				3: (* Wait Z move done *)
				   IF GV_Axes.stAxisZ.bAutoDone THEN
						GV_Axes.stAxisZ.bAutoCmdAbs:=FALSE;
						(*Log*)
							PRG_Log_WM.fbLogWM.M_Write_Log('FB_11_Action_ToolMagazineCheckAll : 2_MoveLocation : 3 : Z move done');
						iSubStep:=4; // Next SubStep
					ELSIF GV_Axes.stAxisZ.stDriveAx8206.AxisRef.Status.Error OR GV_Axes.stAxisZ.stDriveAx8206.AxisRef.Status.ErrorStop OR GV_Axes.stAxisZ.stDriveAx8206.AxisRef.Status.ErrorID<>0 THEN
						bError:=TRUE;
						udiErrorID:=231; // 231 = Step 2 SubStep 3 Error Axis Z 1
						GV_Axes.stAxisZ.bAutoCmdAbs:=FALSE;
						tonTimeout.IN:=FALSE;
						(*Log*)
							PRG_Log_WM.fbLogWM.M_Write_Log('FB_11_Action_ToolMagazineCheckAll : 2_MoveLocation=Error');
							PRG_Log_WM.fbLogWM.M_Write_Log(CONCAT('FB_11_Action_ToolMagazineCheckAll : ErrorID=',UDINT_TO_STRING(udiErrorID)));
						iSubStep:=0; // Stop SubStep
						iStep:=0; // Idle Step
					END_IF

				4: (* Start Y move *)
					GV_Axes.stAxisY.lrAutoPosAbs:=GV_Tool_Magazine.aCheckLocation[iLocation].lrYcoord;
					GV_Axes.stAxisY.bAutoCmdAbs:=TRUE;
					(*Log*)
						PRG_Log_WM.fbLogWM.M_Write_Log('FB_11_Action_ToolMagazineCheckAll : 2_MoveLocation : 4 : Start Y move');
					iSubStep:=5; // Next Step

				5: (* Wait Y move done *)
				   IF GV_Axes.stAxisY.bAutoDone THEN
						GV_Axes.stAxisY.bAutoCmdAbs:=FALSE;
						(*Log*)
							PRG_Log_WM.fbLogWM.M_Write_Log('FB_11_Action_ToolMagazineCheckAll : 2_MoveLocation : 5 : Y move done');
							PRG_Log_WM.fbLogWM.M_Write_Log('FB_11_Action_ToolMagazineCheckAll : 2_MoveLocation->3_Check');
						iSubStep:=0; // End SubStep
						iStep:=3; // Next Step
					ELSIF GV_Axes.stAxisY.stDriveAx8206.AxisRef.Status.Error OR GV_Axes.stAxisY.stDriveAx8206.AxisRef.Status.ErrorStop OR GV_Axes.stAxisY.stDriveAx8206.AxisRef.Status.ErrorID<>0 THEN
						bError:=TRUE;
						udiErrorID:=251; // 251 = Step 2 SubStep 5 Error Axis Y 1
						GV_Axes.stAxisY.bAutoCmdAbs:=FALSE;
						tonTimeout.IN:=FALSE;
						(*Log*)
							PRG_Log_WM.fbLogWM.M_Write_Log('FB_11_Action_ToolMagazineCheckAll : 2_MoveLocation=Error');
							PRG_Log_WM.fbLogWM.M_Write_Log(CONCAT('FB_11_Action_ToolMagazineCheckAll : ErrorID=',UDINT_TO_STRING(udiErrorID)));
						iSubStep:=0; // Stop SubStep
						iStep:=0; // Idle Step
					END_IF

				8: (* Start Y home move *)
					GV_Axes.stAxisY.lrAutoPosAbs:=GV_Tool_Magazine.stManipulator.lrYHome;
					GV_Axes.stAxisY.bAutoCmdAbs:=TRUE;
					(*Log*)
						PRG_Log_WM.fbLogWM.M_Write_Log('FB_11_Action_ToolMagazineCheckAll : 2_MoveLocation : 8 : Start Y home move');
					iSubStep:=9; // Next SubStep

				9: (* Wait Y home move done *)
				   IF GV_Axes.stAxisY.bAutoDone THEN
						GV_Axes.stAxisY.bAutoCmdAbs:=FALSE;
						(*Log*)
							PRG_Log_WM.fbLogWM.M_Write_Log('FB_11_Action_ToolMagazineCheckAll : 2_MoveLocation : 9 : Y home move done');
						iSubStep:=0; // End SubStep
					ELSIF GV_Axes.stAxisY.stDriveAx8206.AxisRef.Status.Error OR GV_Axes.stAxisY.stDriveAx8206.AxisRef.Status.ErrorStop OR GV_Axes.stAxisY.stDriveAx8206.AxisRef.Status.ErrorID<>0 THEN
						bError:=TRUE;
						udiErrorID:=291; // 291 = Step 2 SubStep 9 Error Axis Y 1
						GV_Axes.stAxisY.bAutoCmdAbs:=FALSE;
						tonTimeout.IN:=FALSE;
						(*Log*)
							PRG_Log_WM.fbLogWM.M_Write_Log('FB_11_Action_ToolMagazineCheckAll : 2_MoveLocation=Error');
							PRG_Log_WM.fbLogWM.M_Write_Log(CONCAT('FB_11_Action_ToolMagazineCheckAll : ErrorID=',UDINT_TO_STRING(udiErrorID)));
						iSubStep:=0; // Stop SubStep
						iStep:=0; // Idle Step
					END_IF

				END_CASE
				
				IF tonTimeout.Q THEN
					bError:=TRUE;
					udiErrorID:=299; // 299 = Step 2 Error Timeout 99
					GV_Axes.stAxisX.bAutoCmdAbs:=FALSE;
					GV_Axes.stAxisZ.bAutoCmdAbs:=FALSE;
					GV_Axes.stAxisY.bAutoCmdAbs:=FALSE;
					tonTimeout.IN:=FALSE;
					(*Log*)
						PRG_Log_WM.fbLogWM.M_Write_Log('FB_11_Action_ToolMagazineCheckAll : 2_MoveLocation : Error');
						PRG_Log_WM.fbLogWM.M_Write_Log(CONCAT('FB_11_Action_ToolMagazineCheckAll : ErrorID = ',UDINT_TO_STRING(udiErrorID)));
					iSubStep:=0; // Stop SubStep
					iStep:=0; // Idle Step
				END_IF
	
			3: (* Step 3 = Check Tool presence in Location *)
				(*Conversion*)
					lrToolPresenceRack:=(INT_TO_LREAL(GV_IO.aiToolPresenceRack))*(2/32767); //(0..10V) = (0..32767) = (0..2mm)
				(*Tolerance*)
					IF lrToolPresenceRack>=(lrToolDistance-lrToolDistanceTolerance) AND lrToolPresenceRack<=(lrToolDistance+lrToolDistanceTolerance) THEN
						bToleranceOK:=TRUE;
					ELSE
						bToleranceOK:=FALSE;
					END_IF
				(*Check*)
					IF bToleranceOK THEN
						(*Update*)
							GV_Tool_Magazine.aCheckLocation[iLocation].bToolPresence:=TRUE; // OK
						(*Log*)
							strTextLog:=INT_TO_STRING(GV_IO.aiToolPresenceRack);
							PRG_Log_WM.fbLogWM.M_Write_Log(CONCAT('FB_11_Action_ToolMagazineCheckAll : 3_Check : Sensor in INT = ',strTextLog));
							strTextLog:=LREAL_TO_STRING(lrToolPresenceRack);
							PRG_Log_WM.fbLogWM.M_Write_Log(CONCAT('FB_11_Action_ToolMagazineCheckAll : 3_Check : Sensor in LREAL(mm) = ',strTextLog));
							PRG_Log_WM.fbLogWM.M_Write_Log('FB_11_Action_ToolMagazineCheckAll : 3_Check : Tolerance = OK');						
						bToleranceOK:=FALSE;	
						lrToolPresenceRack:=0.0;
						iStep:=4; // Next Step
					ELSE
						(*Update*)
							GV_Tool_Magazine.aCheckLocation[iLocation].bToolPresence:=FALSE; // NOK
						(*Log*)
							strTextLog:=INT_TO_STRING(GV_IO.aiToolPresenceRack);
							PRG_Log_WM.fbLogWM.M_Write_Log(CONCAT('FB_11_Action_ToolMagazineCheckAll : 3_Check : Sensor in INT = ',strTextLog));
							strTextLog:=LREAL_TO_STRING(lrToolPresenceRack);
							PRG_Log_WM.fbLogWM.M_Write_Log(CONCAT('FB_11_Action_ToolMagazineCheckAll : 3_Check : Sensor in LREAL(mm) = ',strTextLog));
							PRG_Log_WM.fbLogWM.M_Write_Log('FB_11_Action_ToolMagazineCheckAll : 3_Check : Tolerance = NOK');						
						bToleranceOK:=FALSE;	
						lrToolPresenceRack:=0.0;
						iStep:=4; // Next Step
					END_IF
			
			4: (* Step 4 = Next Location Or End *)
				iLocation:=iLocation+1;
				IF iLocation>(GV_Tool_Magazine.iCheckLocationTopSize+GV_Tool_Magazine.iCheckLocationBottomSize) THEN
					(*Log*)
						PRG_Log_WM.fbLogWM.M_Write_Log('FB_11_Action_ToolMagazineCheckAll: End : 4_NextEnd->5_Tunnel');
					iStep:=5; // Next Step = End
				ELSE
					(*Log*)
						PRG_Log_WM.fbLogWM.M_Write_Log('FB_11_Action_ToolMagazineCheckAll : Next : 4_NextEnd->1_Tunnel');
					iStep:=1; // Next Step = Next Location
				END_IF
		(* End Check sequence *)

		5: (* Step 5 = Tunnel passage (if needed) *)
			IF (NOT bTunnelTravel) THEN
				IF GV_Tool_Magazine.stManipulator.ePositionMag=ENUM_Position_Magazine.Top THEN
					bTunnelTravel:=FALSE;
					(*Log*)
						PRG_Log_WM.fbLogWM.M_Write_Log('FB_11_Action_ToolMagazineCheckAll : 5_Tunnel : No Need to Travel');
						PRG_Log_WM.fbLogWM.M_Write_Log('FB_11_Action_ToolMagazineCheckAll : 5_Tunnel->6_PositionHome');
					iSubStep:=0; // For next Step
					iStep:=6; // Next Step
				END_IF	
				IF GV_Tool_Magazine.stManipulator.ePositionMag=ENUM_Position_Magazine.Bottom THEN
					eTunnelMode:=ENUM_Tunnel_MODE.BottomToTop;
					bTunnelTravel:=TRUE;
					(*Log*)
						PRG_Log_WM.fbLogWM.M_Write_Log('FB_11_Action_ToolMagazineCheckAll : 5_Tunnel : Need to Travel Bottom->Top');
				END_IF			
				IF GV_Tool_Magazine.stManipulator.ePositionMag=ENUM_Position_Magazine.Unknow THEN // Manipulator Unknow position
					bError:=TRUE;
					udiErrorID:=501; // 501 = Step 5 Error Tunnel 01
					fbTunnel.bStart:=FALSE;
					bTunnelTravel:=FALSE;
					(*Log*)
						PRG_Log_WM.fbLogWM.M_Write_Log('FB_11_Action_ToolMagazineCheckAll : 5_Tunnel=Error');
						PRG_Log_WM.fbLogWM.M_Write_Log(CONCAT('FB_11_Action_ToolMagazineCheckAll : ErrorID=',UDINT_TO_STRING(udiErrorID)));
					iStep:=0; // Idle Step
				END_IF
			END_IF
			
			IF bTunnelTravel AND (NOT fbTunnel.bStart) AND (NOT fbTunnel.bBusy) THEN // Tunnel Start
				fbTunnel.bStart:=TRUE;
			END_IF
			IF fbTunnel.bDone THEN // Tunnel Done
				fbTunnel.bStart:=FALSE;
				bTunnelTravel:=FALSE;
				(*Log*)
					PRG_Log_WM.fbLogWM.M_Write_Log('FB_11_Action_ToolMagazineCheckAll : 5_Tunnel->6_PositionHome');
				iSubStep:=0; // For next Step
				iStep:=6; // Next Step
			ELSIF fbTunnel.bError THEN // Tunnel Error
				bError:=TRUE;
				udiErrorID:=500+fbTunnel.udiErrorID; // 5xx = Step 5 Error + Error xx fbTunnel
				fbTunnel.bStart:=FALSE;
				bTunnelTravel:=FALSE;
				(*Log*)
					PRG_Log_WM.fbLogWM.M_Write_Log('FB_11_Action_ToolMagazineCheckAll : 5_Tunnel=Error');
					PRG_Log_WM.fbLogWM.M_Write_Log(CONCAT('FB_11_Action_ToolMagazineCheckAll : ErrorID=',UDINT_TO_STRING(udiErrorID)));
				iStep:=0; // Idle Step
			END_IF
			
			IF tonTimeout.Q THEN
				bError:=TRUE;
				udiErrorID:=599; // 599 = Step 5 Error Timeout 99
				fbTunnel.bStart:=FALSE;
				bTunnelTravel:=FALSE;
				tonTimeout.IN:=FALSE;
				(*Log*)
					PRG_Log_WM.fbLogWM.M_Write_Log('FB_11_Action_ToolMagazineCheckAll : 5_Tunnel : Error');
					PRG_Log_WM.fbLogWM.M_Write_Log(CONCAT('FB_11_Action_ToolMagazineCheckAll : ErrorID = ',UDINT_TO_STRING(udiErrorID)));
				iSubStep:=0; // Stop SubStep
				iStep:=0; // Idle Step
			END_IF
				
		6: (* Step 6 = Home Position*)
		
			CASE iSubStep OF //Y->X->Z

				0: (* Start Y home move *)
					GV_Axes.stAxisY.lrAutoPosAbs:=GV_Tool_Magazine.stManipulator.lrYHome;
					GV_Axes.stAxisY.bAutoCmdAbs:=TRUE;
					(*Log*)
						PRG_Log_WM.fbLogWM.M_Write_Log('FB_11_Action_ToolMagazineCheckAll : 6_PositionHome : 0 : Start Y home move');
					iSubStep:=1; // Next Step
				
				1: (* Wait Y home move done *)
					IF GV_Axes.stAxisY.bAutoDone THEN
						GV_Axes.stAxisY.bAutoCmdAbs:=FALSE;
						(*Log*)
							PRG_Log_WM.fbLogWM.M_Write_Log('FB_11_Action_ToolMagazineCheckAll : 6_PositionHome : 1 : Y move done');
						iSubStep:=2; // Next SubStep
					ELSIF GV_Axes.stAxisY.stDriveAx8206.AxisRef.Status.Error OR GV_Axes.stAxisY.stDriveAx8206.AxisRef.Status.ErrorStop OR GV_Axes.stAxisY.stDriveAx8206.AxisRef.Status.ErrorID<>0 THEN
						bError:=TRUE;
						udiErrorID:=611; // 611 = Step 6 SubStep 1 Error Axis Y 1
						GV_Axes.stAxisY.bAutoCmdAbs:=FALSE;
						tonTimeout.IN:=FALSE;
						(*Log*)
							PRG_Log_WM.fbLogWM.M_Write_Log('FB_11_Action_ToolMagazineCheckAll : 6_PositionHome=Error');
							PRG_Log_WM.fbLogWM.M_Write_Log(CONCAT('FB_11_Action_ToolMagazineCheckAll : ErrorID=',UDINT_TO_STRING(udiErrorID)));
						iSubStep:=0; // Stop SubStep
						iStep:=0; // Idle Step
					END_IF
				
				2: (* Start X home move *)
					GV_Axes.stAxisX.lrAutoPosAbs:=GV_Tool_Magazine.stManipulator.lrXHome;
					GV_Axes.stAxisX.bAutoCmdAbs:=TRUE;
					(*Log*)
						PRG_Log_WM.fbLogWM.M_Write_Log('FB_11_Action_ToolMagazineCheckAll : 6_PositionHome : 2 : Start X home move');
					iSubStep:=3; // Next Step
					
				3: (* Wait X home move done *)
					IF GV_Axes.stAxisX.bAutoDone THEN
						GV_Axes.stAxisX.bAutoCmdAbs:=FALSE;
						(*Log*)
							PRG_Log_WM.fbLogWM.M_Write_Log('FB_11_Action_ToolMagazineCheckAll : 6_PositionHome : 3 : X move done');
						iSubStep:=4; // Next SubStep
					ELSIF GV_Axes.stAxisX.stDriveAx8206.AxisRef.Status.Error OR GV_Axes.stAxisX.stDriveAx8206.AxisRef.Status.ErrorStop OR GV_Axes.stAxisX.stDriveAx8206.AxisRef.Status.ErrorID<>0 THEN
						bError:=TRUE;
						udiErrorID:=631; // 631 = Step 6 SubStep 3 Error Axis X 1
						GV_Axes.stAxisX.bAutoCmdAbs:=FALSE;
						tonTimeout.IN:=FALSE;
						(*Log*)
							PRG_Log_WM.fbLogWM.M_Write_Log('FB_11_Action_ToolMagazineCheckAll : 6_PositionHome=Error');
							PRG_Log_WM.fbLogWM.M_Write_Log(CONCAT('FB_11_Action_ToolMagazineCheckAll : ErrorID=',UDINT_TO_STRING(udiErrorID)));
						iSubStep:=0; // Stop SubStep
						iStep:=0; // Idle Step
					END_IF
				
				4: (* Start Z home move *)
					GV_Axes.stAxisZ.lrAutoPosAbs:=GV_Tool_Magazine.stManipulator.lrZHome;
					GV_Axes.stAxisZ.bAutoCmdAbs:=TRUE;
					(*Log*)
						PRG_Log_WM.fbLogWM.M_Write_Log('FB_11_Action_ToolMagazineCheckAll : 6_PositionHome : 4 : Start X home move');
					iSubStep:=5; // Next Step
					
				5: (* Wait Z home move done *)
					IF GV_Axes.stAxisZ.bAutoDone THEN
						GV_Axes.stAxisZ.bAutoCmdAbs:=FALSE;
						(*Log*)
							PRG_Log_WM.fbLogWM.M_Write_Log('FB_11_Action_ToolMagazineCheckAll : 6_PositionHome : 5 : Y move done');
							PRG_Log_WM.fbLogWM.M_Write_Log('FB_11_Action_ToolMagazineCheckAll : 6_PositionHome->0_Idle');
						tonTimeout.IN:=FALSE;
						iSubStep:=0; // End SubStep
						iStep:=0; // End Step
						bDone:=TRUE;
						bBusy:=FALSE;
					ELSIF GV_Axes.stAxisZ.stDriveAx8206.AxisRef.Status.Error OR GV_Axes.stAxisZ.stDriveAx8206.AxisRef.Status.ErrorStop OR GV_Axes.stAxisZ.stDriveAx8206.AxisRef.Status.ErrorID<>0 THEN
						bError:=TRUE;
						udiErrorID:=651; // 651 = Step 6 SubStep 5 Error Axis Z 1
						GV_Axes.stAxisZ.bAutoCmdAbs:=FALSE;
						tonTimeout.IN:=FALSE;
						(*Log*)
							PRG_Log_WM.fbLogWM.M_Write_Log('FB_11_Action_ToolMagazineCheckAll : 6_PositionHome=Error');
							PRG_Log_WM.fbLogWM.M_Write_Log(CONCAT('FB_11_Action_ToolMagazineCheckAll : ErrorID=',UDINT_TO_STRING(udiErrorID)));
						iSubStep:=0; // Stop SubStep
						iStep:=0; // Idle Step
					END_IF
					
			END_CASE
				
			IF tonTimeout.Q AND tonTimeout.PT<>T#0S THEN
				bError:=TRUE;
				udiErrorID:=699; // 699 = Step 6 Error Timeout 99
				GV_Axes.stAxisX.bAutoCmdAbs:=FALSE;
				GV_Axes.stAxisZ.bAutoCmdAbs:=FALSE;
				GV_Axes.stAxisY.bAutoCmdAbs:=FALSE;
				tonTimeout.IN:=FALSE;
				(*Log*)
					PRG_Log_WM.fbLogWM.M_Write_Log('FB_11_Action_ToolMagazineCheckAll : 6_PositionHome : Error');
					PRG_Log_WM.fbLogWM.M_Write_Log(CONCAT('FB_11_Action_ToolMagazineCheckAll : ErrorID = ',UDINT_TO_STRING(udiErrorID)));
				iSubStep:=0; // Stop SubStep
				iStep:=0; // Idle Step
			END_IF

	END_CASE

END_FUNCTION_BLOCK

// ---- 08_Cycle/03_POUs/02_FBs/FB_200_Action_HomePosition.TcPOU
FUNCTION_BLOCK FB_200_Action_HomePosition
VAR_INPUT
	(** SETUP ST **)
		
	(** SETUP TIME **)
		(*Tunnel*)
			tTunnelTimeout : TIME ; // Value of the timeout for travel the tunnel
		(* Step x *)
			tMovexTimeout : TIME ; // Value of the timeout for Step x

	(** SETUP LREAL **)

	(** SETUP FLAG **)
			
	(** PROCESS FLAG **)
	    bInit : BOOL ; // Init the Fb
	    bStart : BOOL ; // Start the Fb
END_VAR
VAR_OUTPUT
	(** PROCESS UDINT **)
		udiErrorID : UDINT ; // Fb Error ID
		
	(** PROCESS FLAG **)
		bBusy  : BOOL ; // Fb is Busy
		bDone  : BOOL ; // Fb is Done
		bError : BOOL ; // Fb in Error
END_VAR
VAR_IN_OUT
END_VAR	
VAR
	(** SETUP ENUM **)
		(*Tunnel*)
			eTunnelMode : ENUM_Tunnel_Mode; // Tunnel mode for travel (fbTunnel)

	(** SETUP TIME **)
	
	(** SETUP FLAG **)
		
	(** PROCESS STRING **)
		strTextLog : STRING ; // Text to Log
		
	(** PROCESS LREAL **)
		
	(** PROCESS INT **)
		iStep  : INT := 0 ; // Step of the Fb
		iSubStep : INT := 0 ; // SubStep of the Fb
		iPrevStep : INT := 0 ; // Previous Step of the Fb
		iPrevSubStep : INT := 0 ; // Previous Subtep of the Fb
		
	(** PROCESS FLAG + R_TRIG **)
		rtInit : R_TRIG ; // FB Init at rising edge
		rtStart : R_TRIG ; // FB Start at rising edge
		(*Tunnel*)
			bTunnelTravel : BOOL ; // Need to travel the tunnel
				
	(** FB **)
		(*Tunnel*)
			fbTunnel : FB_Manipulator_Tunnel ;
		(* Step x *)
			tonTimeoutMovex : TON ; // TON timeout for the Step x
END_VAR

//-----------------------------------------------------------------------------------------
//
//                  			FB_200_Action_HomePosition
//
//		ESSAI		Management of move to home position (Manipulator only)
//-----------------------------------------------------------------------------------------
//
//Auteur: G.GOETZ
//Création: 01.04.2026
//Dernière modification : 01.04.2026 (G.GOETZ)
//       			
//-----------------------------------------------------------------------------------------
//
//     							Liste des modifications  	
//
// 01.04.2026 (G.GOETZ) -> Création		
//-----------------------------------------------------------------------------------------

(** FB CALL **)
	rtInit(CLK:=bInit);
	rtStart(CLK:=bStart);
		
	tonTimeoutMovex();
	fbTunnel( // Call Tunnel travel
			eTunnelMode:=eTunnelMode,
			tTimeout:=tTunnelTimeout
			);

(** INIT **)
	IF (rtinit.Q OR bInit) AND (NOT bStart) THEN
		bBusy:=FALSE;
		bDone:=FALSE;
		bError:=FALSE;
		udiErrorID:=0;
		iStep:=0;
		iSubStep:=0;
		bInit:=FALSE;
	END_IF

(** STEPS **)
    CASE iStep OF
		
        0: (* Step 0 = Idle + Check *)
            bBusy:=FALSE;
            bDone:=FALSE;
			bError:=FALSE;
			udiErrorID:=0;
			iSubStep:=0;
			
			tonTimeoutMovex.IN:=FALSE;
			
			bTunnelTravel:=FALSE;
			
			(* Idle->Start *)
				IF rtStart.Q AND (NOT bInit) THEN
					bBusy:=TRUE;
					(*Log*)
						PRG_Log_WM.fbLogWM.M_Write_Log('FB_200_Action_HomePosition : 0_Idle : Manipulator to Home Position');
						PRG_Log_WM.fbLogWM.M_Write_Log('FB_200_Action_HomePosition : 0_Idle->1_Tunnel');
					iStep:=1;
				END_IF
				
		1: (* Step 1 = Tunnel passage (if needed) *)
			IF (NOT bTunnelTravel) THEN
				IF GV_Tool_Magazine.stManipulator.ePositionMag=ENUM_Position_Magazine.Top THEN
					bTunnelTravel:=FALSE;
					(*Log*)
						PRG_Log_WM.fbLogWM.M_Write_Log('FB_200_Action_HomePosition : 1_Tunnel : No Need to Travel');
						PRG_Log_WM.fbLogWM.M_Write_Log('FB_200_Action_HomePosition : 1_Tunnel->2_MoveHome');
					iStep:=2; // Next Step
				END_IF	
				IF GV_Tool_Magazine.stManipulator.ePositionMag=ENUM_Position_Magazine.Bottom THEN
					eTunnelMode:=ENUM_Tunnel_MODE.BottomToTop;
					bTunnelTravel:=TRUE;
					(*Log*)
						PRG_Log_WM.fbLogWM.M_Write_Log('FB_200_Action_HomePosition : 1_Tunnel : Need to Travel Bottom->Top');
				END_IF			
				IF GV_Tool_Magazine.stManipulator.ePositionMag=ENUM_Position_Magazine.Unknow THEN // Manipulator Unknow position
					bError:=TRUE;
					udiErrorID:=101; // 101 = Step 1 Error Tunnel 01
					fbTunnel.bStart:=FALSE;
					bTunnelTravel:=FALSE;
					(*Log*)
						PRG_Log_WM.fbLogWM.M_Write_Log('FB_200_Action_HomePosition : 1_Tunnel=Error');
						PRG_Log_WM.fbLogWM.M_Write_Log(CONCAT('FB_200_Action_HomePosition : ErrorID=',UDINT_TO_STRING(udiErrorID)));
					iStep:=0; // Idle Step
				END_IF
			END_IF
			
			IF bTunnelTravel AND (NOT fbTunnel.bStart) AND (NOT fbTunnel.bBusy) THEN // Tunnel Start
				fbTunnel.bStart:=TRUE;
			END_IF
			IF fbTunnel.bDone THEN // Tunnel Done
				fbTunnel.bStart:=FALSE;
				bTunnelTravel:=FALSE;
				(*Log*)
					PRG_Log_WM.fbLogWM.M_Write_Log('FB_200_Action_HomePosition : 1_Tunnel->2_MoveHome');
				iStep:=2; // Next Step
			ELSIF fbTunnel.bError THEN // Tunnel Error
				bError:=TRUE;
				udiErrorID:=100+fbTunnel.udiErrorID; // 1xx = Step 1 Error + Error xx fbTunnel
				fbTunnel.bStart:=FALSE;
				bTunnelTravel:=FALSE;
				(*Log*)
					PRG_Log_WM.fbLogWM.M_Write_Log('FB_200_Action_HomePosition : 1_Tunnel=Error');
					PRG_Log_WM.fbLogWM.M_Write_Log(CONCAT('FB_200_Action_HomePosition : ErrorID=',UDINT_TO_STRING(udiErrorID)));
				iStep:=0; // Idle Step
			END_IF
			
		2: (* Step 2 = Move the manipulator to Home (Y->Z->X) *)
			tonTimeoutMovex.PT:=tMovexTimeout;
			tonTimeoutMovex.IN:=TRUE;
			
			CASE iSubStep OF
        
				0: (* Start Y move *)
					GV_Axes.stAxisY.lrAutoPosAbs:=GV_Tool_Magazine.stManipulator.lrYHome;
					GV_Axes.stAxisY.bAutoCmdAbs:=TRUE;
					(*Log*)
						PRG_Log_WM.fbLogWM.M_Write_Log('FB_200_Action_HomePosition : 2_MoveHome : 0 : Start Y move');
					iSubStep:=1; // Next SubStep

				1: (* Wait Y move done *)
				   IF GV_Axes.stAxisY.bAutoDone THEN
						GV_Axes.stAxisY.bAutoCmdAbs:=FALSE;
						(*Log*)
							PRG_Log_WM.fbLogWM.M_Write_Log('FB_200_Action_HomePosition : 2_MoveHome : 1 : Y move done');
						iSubStep:=2; // Next SubStep
					ELSIF GV_Axes.stAxisY.stDriveAx8206.AxisRef.Status.Error OR GV_Axes.stAxisY.stDriveAx8206.AxisRef.Status.ErrorStop OR GV_Axes.stAxisY.stDriveAx8206.AxisRef.Status.ErrorID<>0 THEN
						bError:=TRUE;
						udiErrorID:=211; // 211 = Step 2 SubStep 1 Error Axis Y 1
						GV_Axes.stAxisY.bAutoCmdAbs:=FALSE;
						tonTimeoutMovex.IN:=FALSE;
						(*Log*)
							PRG_Log_WM.fbLogWM.M_Write_Log('FB_200_Action_HomePosition : 2_MoveHome=Error');
							PRG_Log_WM.fbLogWM.M_Write_Log(CONCAT('FB_200_Action_HomePosition : ErrorID=',UDINT_TO_STRING(udiErrorID)));
						iSubStep:=0; // Stop SubStep
						iStep:=0; // Idle Step
					END_IF
				
				2: (* Start Z move *)
					GV_Axes.stAxisZ.lrAutoPosAbs:=GV_Tool_Magazine.stManipulator.lrZHome;
					GV_Axes.stAxisZ.bAutoCmdAbs:=TRUE;
					(*Log*)
						PRG_Log_WM.fbLogWM.M_Write_Log('FB_200_Action_HomePosition : 2_MoveHome : 2 : Start Z move');
					iSubStep:=3; // Next SubStep

				3: (* Wait Z move done *)
				   IF GV_Axes.stAxisZ.bAutoDone THEN
						GV_Axes.stAxisZ.bAutoCmdAbs:=FALSE;
						(*Log*)
							PRG_Log_WM.fbLogWM.M_Write_Log('FB_200_Action_HomePosition : 2_MoveHome : 3 : Z move done');
						iSubStep:=4; // Next SubStep
					ELSIF GV_Axes.stAxisZ.stDriveAx8206.AxisRef.Status.Error OR GV_Axes.stAxisZ.stDriveAx8206.AxisRef.Status.ErrorStop OR GV_Axes.stAxisZ.stDriveAx8206.AxisRef.Status.ErrorID<>0 THEN
						bError:=TRUE;
						udiErrorID:=231; // 231 = Step 2 SubStep 3 Error Axis Z 1
						GV_Axes.stAxisZ.bAutoCmdAbs:=FALSE;
						tonTimeoutMovex.IN:=FALSE;
						(*Log*)
							PRG_Log_WM.fbLogWM.M_Write_Log('FB_200_Action_HomePosition : 2_MoveHome=Error');
							PRG_Log_WM.fbLogWM.M_Write_Log(CONCAT('FB_200_Action_HomePosition : ErrorID=',UDINT_TO_STRING(udiErrorID)));
						iSubStep:=0; // Stop SubStep
						iStep:=0; // Idle Step
					END_IF

				4: (* Start X move *)
					GV_Axes.stAxisX.lrAutoPosAbs:=GV_Tool_Magazine.stManipulator.lrXHome;
					GV_Axes.stAxisX.bAutoCmdAbs:=TRUE;
					(*Log*)
						PRG_Log_WM.fbLogWM.M_Write_Log('FB_200_Action_HomePosition : 2_MoveHome : 4 : Start X move');
					iSubStep:=5; // Next Step

				5: (* Wait X move done *)
				   IF GV_Axes.stAxisX.bAutoDone THEN
						GV_Axes.stAxisX.bAutoCmdAbs:=FALSE;
						tonTimeoutMovex.IN:=FALSE;
						(*Log*)
							PRG_Log_WM.fbLogWM.M_Write_Log('FB_200_Action_HomePosition : 2_MoveHome : 5 : X move done');
							PRG_Log_WM.fbLogWM.M_Write_Log('FB_200_Action_HomePosition : 2_MoveHome->0_Idle');
						iSubStep:=0; // End SubStep
						iStep:=0; // End Step
						bDone:=TRUE;
						bBusy:=FALSE;
					ELSIF GV_Axes.stAxisX.stDriveAx8206.AxisRef.Status.Error OR GV_Axes.stAxisX.stDriveAx8206.AxisRef.Status.ErrorStop OR GV_Axes.stAxisX.stDriveAx8206.AxisRef.Status.ErrorID<>0 THEN
						bError:=TRUE;
						udiErrorID:=251; // 251 = Step 2 SubStep 5 Error Axis X 1
						GV_Axes.stAxisX.bAutoCmdAbs:=FALSE;
						tonTimeoutMovex.IN:=FALSE;
						(*Log*)
							PRG_Log_WM.fbLogWM.M_Write_Log('FB_200_Action_HomePosition : 2_MoveHome=Error');
							PRG_Log_WM.fbLogWM.M_Write_Log(CONCAT('FB_200_Action_HomePosition : ErrorID=',UDINT_TO_STRING(udiErrorID)));
						iSubStep:=0; // Stop SubStep
						iStep:=0; // Idle Step
					END_IF
					
			END_CASE	
		
			IF tonTimeoutMovex.Q AND tonTimeoutMovex.PT<>T#0S THEN // Timeout 
				bError:=TRUE;
				udiErrorID:=299; // 299 = Step 2 Error Timeout 99
				GV_Axes.stAxisZ.bAutoCmdAbs:=FALSE;
				GV_Axes.stAxisX.bAutoCmdAbs:=FALSE;
				GV_Axes.stAxisY.bAutoCmdAbs:=FALSE;
				tonTimeoutMovex.IN:=FALSE;
				(*Log*)
					PRG_Log_WM.fbLogWM.M_Write_Log('FB_200_Action_HomePosition : 2_MoveHome=Error');
					PRG_Log_WM.fbLogWM.M_Write_Log(CONCAT('FB_200_Action_HomePosition : ErrorID=',UDINT_TO_STRING(udiErrorID)));
				iSubStep:=0;
				iStep:=0;
			END_IF
				
	END_CASE

END_FUNCTION_BLOCK

// ---- 08_Cycle/03_POUs/02_FBs/FB_202_Action_PickPlaceToolMag.TcPOU
FUNCTION_BLOCK FB_202_Action_PickPlaceToolMag
VAR_INPUT
	(** SETUP ST **)
		stToolLocation : ST_Tool_Location ; // Tool_Location structure of the Tool to Go
		
	(** SETUP TIME **)
		(*Manipulator Gripper mvmnt*)
			tMouvementGripperOpen : TIME ; // Value of the manipulator gripper open mouvement duration
			tMouvementGripperClose : TIME ; // Value of the manipulator gripper close mouvement duration
		(*Tunnel*)
			tTunnelTimeout : TIME ; // Value of the timeout for travel the tunnel
		(* Step x *)
			tMovexTimeout : TIME ; // Value of the timeout for Step x

	(** SETUP LREAL **)
		lrToolDistance : LREAL ; // Theoretical distance in mm for tool presence
		
		lrOffsetX : LREAL ;
		lrOffsetY : LREAL ;

	(** SETUP FLAG **)
		bCheckSensorManipulatorGripper : BOOL ; // Check the manipulator gripper sensor at the beginning
		(*Gripper*)
			bCheckSensorGripperOpen : BOOL ; // Check the manipulator gripper sensor after open
			bCheckSensorGripperClose : BOOL ; // Check the manipulator gripper sensor after close	
			
	(** PROCESS FLAG **)
	    bInit : BOOL ; // Init the Fb
	    bStart : BOOL ; // Start the Fb
END_VAR
VAR_OUTPUT
	(** PROCESS UUDINT **)
		udiErrorID : UDINT ; // Fb Error ID
		
	(** PROCESS FLAG **)
		bBusy  : BOOL ; // Fb is Busy
		bDone  : BOOL ; // Fb is Done
		bError : BOOL ; // Fb in Error
END_VAR
VAR_IN_OUT
END_VAR	
VAR
	(** SETUP ENUM **)
		(*Manipulator Gripper mvmnt*)
			eGripperMode : ENUM_Gripper_Mode; // Gripper mode for gripper mouvement (fbGripper)
		(*Tunnel*)
			eTunnelMode : ENUM_Tunnel_Mode; // Tunnel mode for travel (fbTunnel)

	(** SETUP TIME **)
		(*Manipulator Gripper mvmnt*)
			tGripperTime : TIME ; // Mouvement duration for gripper mouvement (fbGripper)
			
	(** SETUP FLAG **)
		(*Manipulator Gripper mvmnt*)
			bGripperSensor : BOOL ; // Sensor check for gripper mouvement (fbGripper)
			
	(** PROCESS STRING **)
		strTextLog : STRING ; // Text to Log
		
	(** PROCESS LREAL **)
		
	(** PROCESS INT **)
		iStep  : INT := 0 ; // Step of the Fb
		iSubStep : INT := 0 ; // SubStep of the Fb
		iPrevStep : INT := 0 ; // Previous Step of the Fb
		iPrevSubStep : INT := 0 ; // Previous Subtep of the Fb
		
	(** PROCESS FLAG + R_TRIG **)
		rtInit : R_TRIG ; // FB Init at rising edge
		rtStart : R_TRIG ; // FB Start at rising edge
		(*Tunnel*)
			bTunnelTravel : BOOL ; // Need to travel the tunnel
				
	(** FB **)
		(*Gripper*)
			fbGripper : FB_Manipulator_Gripper ;
		(*Tunnel*)
			fbTunnel : FB_Manipulator_Tunnel ;
		(* Step x *)
			tonTimeoutMovex : TON ; // TON timeout for the Step x

END_VAR

//-----------------------------------------------------------------------------------------
//
//                  			FB_202_Action_PickTool
//
//		ESSAI		Management of pick tool in magazine (Manipulator only)
//-----------------------------------------------------------------------------------------
//
//Auteur: G.GOETZ
//Création: 05.04.2026
//Dernière modification : 05.04.2026 (G.GOETZ)
//       			
//-----------------------------------------------------------------------------------------
//
//     							Liste des modifications  	
//
// 05.04.2026 (G.GOETZ) -> Création		
//-----------------------------------------------------------------------------------------

(** FB CALL **)
	rtInit(CLK:=bInit);
	rtStart(CLK:=bStart);

	tonTimeoutMovex();
	fbGripper( // Call Griper mouvement
			eGripperMode:=eGripperMode,
			tMouvementDuration:=tGripperTime,
			bSensorCheck:=bGripperSensor
			);
	fbTunnel( // Call Tunnel travel
			eTunnelMode:=eTunnelMode,
			tTimeout:=tTunnelTimeout
			);

(** INIT **)
	IF (rtinit.Q OR bInit) AND (NOT bStart) THEN
		bBusy:=FALSE;
		bDone:=FALSE;
		bError:=FALSE;
		udiErrorID:=0;
		iStep:=0;
		iSubStep:=0;
		bInit:=FALSE;
	END_IF

(** STEPS **)
    CASE iStep OF
		
        0: (* Step 0 = Idle + Check *)
            bBusy:=FALSE;
            bDone:=FALSE;
			bError:=FALSE;
			udiErrorID:=0;
			iSubStep:=0;
			tonTimeoutMovex.IN:=FALSE;
			bTunnelTravel:=FALSE;
			(* Idle->Start *)
				IF rtStart.Q AND (NOT bInit) THEN
					bBusy:=TRUE;
					(*Log*)
						(*Location*)
							strTextLog:=INT_TO_STRING(stToolLocation.iAbsLocationNumber);
							PRG_Log_WM.fbLogWM.M_Write_Log(CONCAT('FB_202_Action_PickPlaceToolMag : 0_Idle : Tool Location Abs = ',strTextLog));
							strTextLog:=INT_TO_STRING(stToolLocation.iRelLocationNumber);
							PRG_Log_WM.fbLogWM.M_Write_Log(CONCAT('FB_202_Action_PickPlaceToolMag : 0_Idle : Tool Location Rel = ',strTextLog));
							strTextLog:=DINT_TO_STRING(stToolLocation.stToolParam.Number);
							PRG_Log_WM.fbLogWM.M_Write_Log(CONCAT('FB_202_Action_PickPlaceToolMag : 0_Idle : Tool Number = ',strTextLog));
						(*Sensor Check Manipulator*)
							IF bCheckSensorManipulatorGripper THEN
								strTextLog:='With';
							ELSE
								strTextLog:='Without';
							END_IF
							PRG_Log_WM.fbLogWM.M_Write_Log(CONCAT('FB_202_Action_PickPlaceToolMag : 0_Idle : Sensor Manipulator memory Check = ',strTextLog));
						(*Tool Location Distance*)
							strTextLog:=LREAL_TO_STRING(lrToolDistance);
							PRG_Log_WM.fbLogWM.M_Write_Log(CONCAT('FB_202_Action_PickPlaceToolMag : 0_Idle : Tool Distance = ',strTextLog));
						(*Timeout Step X*)
							strTextLog:=TIME_TO_STRING(tMovexTimeout);
							PRG_Log_WM.fbLogWM.M_Write_Log(CONCAT('FB_202_Action_PickPlaceToolMag : 0_Idle : Timeout Step : X = ',strTextLog));

					(*Check manipulator memory/sensor*)
						IF (NOT GV_Tool_Magazine.stManipulator.bToolPresenceMemory) THEN
							(*Log*)
								PRG_Log_WM.fbLogWM.M_Write_Log('FB_202_Action_PickPlaceToolMag : 0_Idle : Manipulator memory Check = OK');
								
							(*Check manipulator gripper*)
// 								IF (NOT GV_CNC.stFanucData.stMagazineCNC.boOpenManipulatorGripper) THEN // Gripper close
// 									(*Log*)
// 										PRG_Log_WM.fbLogWM.M_Write_Log('FB_202_Action_PickPlaceToolMag : 0_Idle : Manipulator gripper Check = OK');
// 										PRG_Log_WM.fbLogWM.M_Write_Log('FB_202_Action_PickPlaceToolMag : 0_Idle : Manipulator gripper = Close');
// 								ELSE
// 									bError:=TRUE;
// 									udiErrorID:=003; // 003 = Step 0 Error Manipulator Gripper Check 03
// 									(*Log*)
// 										PRG_Log_WM.fbLogWM.M_Write_Log('FB_202_Action_PickPlaceToolMag : 0_Idle : Manipulator gripper Check = NOK');
// 										PRG_Log_WM.fbLogWM.M_Write_Log('FB_202_Action_PickPlaceToolMag : 0_Idle : Manipulator gripper = Open');
// 										PRG_Log_WM.fbLogWM.M_Write_Log('FB_202_Action_PickPlaceToolMag : 0_Idle=Error');
// 										PRG_Log_WM.fbLogWM.M_Write_Log(CONCAT('FB_202_Action_PickPlaceToolMag : ErrorID=',UDINT_TO_STRING(udiErrorID)));
// 									iStep:=0; // Idle Step
// 								END_IF
								
								IF bCheckSensorManipulatorGripper THEN
									IF (NOT GV_IO.diToolPresenceCone) THEN
										(*Log*)
											PRG_Log_WM.fbLogWM.M_Write_Log('FB_202_Action_PickPlaceToolMag : 0_Idle : Manipulator sensor Check = FALSE = OK');
											PRG_Log_WM.fbLogWM.M_Write_Log('FB_202_Action_PickPlaceToolMag : 0_Idle->1_Tunnel');
										iStep:=1;
									ELSE
										bError:=TRUE;
										udiErrorID:=002; // 002 = Step 0 Error Manipulator Sensor Check 02
										(*Log*)
											PRG_Log_WM.fbLogWM.M_Write_Log('FB_202_Action_PickPlaceToolMag : 0_Idle : Manipulator sensor Check = TRUE = NOK');
											PRG_Log_WM.fbLogWM.M_Write_Log('FB_202_Action_PickPlaceToolMag : 0_Idle=Error');
											PRG_Log_WM.fbLogWM.M_Write_Log(CONCAT('FB_202_Action_PickPlaceToolMag : ErrorID=',UDINT_TO_STRING(udiErrorID)));
										iStep:=0; // Idle Step
									END_IF
								ELSE
									(*Log*)
										PRG_Log_WM.fbLogWM.M_Write_Log('FB_202_Action_PickPlaceToolMag : 0_Idle : Manipulator sensor Check : Not controlled');
										PRG_Log_WM.fbLogWM.M_Write_Log('FB_202_Action_PickPlaceToolMag : 0_Idle->1_Tunnel');
									iStep:=1;
								END_IF
						ELSE
							bError:=TRUE;
							udiErrorID:=001; // 001 = Step 0 Error Manipulator Memory Check 01
							(*Log*)
								PRG_Log_WM.fbLogWM.M_Write_Log('FB_202_Action_PickPlaceToolMag : 0_Idle : Manipulator memory Check = NOK');
								PRG_Log_WM.fbLogWM.M_Write_Log('FB_202_Action_PickPlaceToolMag : 0_Idle : Manipulator memory = Presence');
								strTextLog:=INT_TO_STRING(GV_Tool_Magazine.stManipulator.iAbsLocationNumberMemory);
								PRG_Log_WM.fbLogWM.M_Write_Log(CONCAT('FB_202_Action_PickPlaceToolMag : 0_Idle : Manipulator memory Location Number Abs = ',strTextLog));
								strTextLog:=INT_TO_STRING(GV_Tool_Magazine.stManipulator.iRelLocationNumberMemory);
								PRG_Log_WM.fbLogWM.M_Write_Log(CONCAT('FB_202_Action_PickPlaceToolMag : 0_Idle : Manipulator memory Location Number Rel = ',strTextLog));
								PRG_Log_WM.fbLogWM.M_Write_Log('FB_202_Action_PickPlaceToolMag : 0_Idle=Error');
								PRG_Log_WM.fbLogWM.M_Write_Log(CONCAT('FB_202_Action_PickPlaceToolMag : ErrorID=',UDINT_TO_STRING(udiErrorID)));
							iStep:=0; // Idle Step
						END_IF
				END_IF
				
		1: (* Step 1 = Tunnel passage (if needed) *)
						
			IF (NOT bTunnelTravel) THEN
				IF (stToolLocation.ePositionMag=ENUM_Position_Magazine.Bottom AND GV_Tool_Magazine.stManipulator.ePositionMag=ENUM_Position_Magazine.Bottom) OR (stToolLocation.ePositionMag=ENUM_Position_Magazine.Top AND GV_Tool_Magazine.stManipulator.ePositionMag=ENUM_Position_Magazine.Top) THEN
					bTunnelTravel:=FALSE;
					(*Log*)
						PRG_Log_WM.fbLogWM.M_Write_Log('FB_202_Action_PickPlaceToolMag : 1_Tunnel : No Need to Travel');
						PRG_Log_WM.fbLogWM.M_Write_Log('FB_202_Action_PickPlaceToolMag : 1_Tunnel->2_AboveLocation');
					iStep:=2; // Next Step
				END_IF	
				IF stToolLocation.ePositionMag=ENUM_Position_Magazine.Bottom AND GV_Tool_Magazine.stManipulator.ePositionMag=ENUM_Position_Magazine.Top THEN
					eTunnelMode:=ENUM_Tunnel_MODE.TopToBottom;
					bTunnelTravel:=TRUE;
					(*Log*)
						PRG_Log_WM.fbLogWM.M_Write_Log('FB_202_Action_PickPlaceToolMag : 1_Tunnel : Need to Travel Top->Bottom');
				END_IF
				IF stToolLocation.ePositionMag=ENUM_Position_Magazine.Top AND GV_Tool_Magazine.stManipulator.ePositionMag=ENUM_Position_Magazine.Bottom THEN
					eTunnelMode:=ENUM_Tunnel_MODE.BottomToTop;
					bTunnelTravel:=TRUE;
					(*Log*)
						PRG_Log_WM.fbLogWM.M_Write_Log('FB_202_Action_PickPlaceToolMag : 1_Tunnel : Need to Travel Bottom->Top');
				END_IF			
				IF stToolLocation.ePositionMag<>ENUM_Position_Magazine.Unknow AND GV_Tool_Magazine.stManipulator.ePositionMag=ENUM_Position_Magazine.Unknow THEN // Manipulator Unknow position
					bError:=TRUE;
					udiErrorID:=101; // 101 = Step 1 Error Tunnel 01
					bTunnelTravel:=FALSE;
					(*Log*)
						PRG_Log_WM.fbLogWM.M_Write_Log('FB_202_Action_PickPlaceToolMag : 1_Tunnel=Error');
						PRG_Log_WM.fbLogWM.M_Write_Log(CONCAT('FB_202_Action_PickPlaceToolMag : ErrorID=',UDINT_TO_STRING(udiErrorID)));
					iStep:=0; // Idle Step
				END_IF
				IF stToolLocation.ePositionMag=ENUM_Position_Magazine.Unknow AND GV_Tool_Magazine.stManipulator.ePositionMag<>ENUM_Position_Magazine.Unknow THEN // ToolLocation Unknow position
					bError:=TRUE;
					udiErrorID:=102; // 102 = Step 1 Error Tunnel 02
					bTunnelTravel:=FALSE;
					(*Log*)
						PRG_Log_WM.fbLogWM.M_Write_Log('FB_202_Action_PickPlaceToolMag : 1_Tunnel=Error');
						PRG_Log_WM.fbLogWM.M_Write_Log(CONCAT('FB_202_Action_PickPlaceToolMag : ErrorID=',UDINT_TO_STRING(udiErrorID)));
					iStep:=0; // Idle Step
				END_IF
				IF stToolLocation.ePositionMag=ENUM_Position_Magazine.Unknow AND GV_Tool_Magazine.stManipulator.ePositionMag=ENUM_Position_Magazine.Unknow THEN // ToolLocation AND Manipulator Unknow position
					bError:=TRUE;
					udiErrorID:=103; // 103 = Step 1 Error Tunnel 03
					bTunnelTravel:=FALSE;
					(*Log*)
						PRG_Log_WM.fbLogWM.M_Write_Log('FB_202_Action_PickPlaceToolMag : 1_Tunnel=Error');
						PRG_Log_WM.fbLogWM.M_Write_Log(CONCAT('FB_202_Action_PickPlaceToolMag : ErrorID=',UDINT_TO_STRING(udiErrorID)));
					iStep:=0; // Idle Step
				END_IF
			END_IF
			
			IF bTunnelTravel AND (NOT fbTunnel.bStart) AND (NOT fbTunnel.bBusy) THEN // Tunnel Start
				fbTunnel.bStart:=TRUE;
			END_IF
			IF fbTunnel.bDone THEN // Tunnel Done
				fbTunnel.bStart:=FALSE;
				bTunnelTravel:=FALSE;
				(*Log*)
					PRG_Log_WM.fbLogWM.M_Write_Log('FB_202_Action_PickPlaceToolMag : 1_Tunnel->2_AboveLocation');
				iSubStep:=0; // For next Step
				iStep:=2; // Next Step
			ELSIF fbTunnel.bError THEN // Tunnel Error
				bError:=TRUE;
				udiErrorID:=100+fbTunnel.udiErrorID; // 1xx = Step 1 Error + Error xx fbTunnel
				fbTunnel.bStart:=FALSE;
				bTunnelTravel:=FALSE;
				(*Log*)
					PRG_Log_WM.fbLogWM.M_Write_Log('FB_202_Action_PickPlaceToolMag : 1_Tunnel=Error');
					PRG_Log_WM.fbLogWM.M_Write_Log(CONCAT('FB_202_Action_PickPlaceToolMag : ErrorID=',UDINT_TO_STRING(udiErrorID)));
				iStep:=0; // Idle Step
			END_IF
		
		2: (* Step 2 = Move the manipulator above the tool/location (Yhome->Zoffset->X->Y) *)
			tonTimeoutMovex.PT:=tMovexTimeout;
			tonTimeoutMovex.IN:=TRUE;
			
			CASE iSubStep OF
        
				0: (* Start Y move *)
					GV_Axes.stAxisY.lrAutoPosAbs:=GV_Tool_Magazine.stManipulator.lrYHome;
					GV_Axes.stAxisY.bAutoCmdAbs:=TRUE;
					(*Log*)
						PRG_Log_WM.fbLogWM.M_Write_Log('FB_202_Action_PickPlaceToolMag : 2_AboveLocation : 0 : Start Y move home');
					iSubStep:=1; // Next SubStep

				1: (* Wait Y move done *)
				   IF GV_Axes.stAxisY.bAutoDone THEN
						GV_Axes.stAxisY.bAutoCmdAbs:=FALSE;
						(*Log*)
							PRG_Log_WM.fbLogWM.M_Write_Log('FB_202_Action_PickPlaceToolMag : 2_AboveLocation : 1 : Y move home done');
						iSubStep:=2; // Next SubStep
					ELSIF GV_Axes.stAxisY.stDriveAx8206.AxisRef.Status.Error OR GV_Axes.stAxisY.stDriveAx8206.AxisRef.Status.ErrorStop OR GV_Axes.stAxisY.stDriveAx8206.AxisRef.Status.ErrorID<>0 THEN
						bError:=TRUE;
						udiErrorID:=211; // 211 = Step 2 SubStep 1 Error Axis Y 1
						GV_Axes.stAxisY.bAutoCmdAbs:=FALSE;
						tonTimeoutMovex.IN:=FALSE;
						(*Log*)
							PRG_Log_WM.fbLogWM.M_Write_Log('FB_202_Action_PickPlaceToolMag : 2_AboveLocation=Error');
							PRG_Log_WM.fbLogWM.M_Write_Log(CONCAT('FB_202_Action_PickPlaceToolMag : ErrorID=',UDINT_TO_STRING(udiErrorID)));
						iSubStep:=0; // Stop SubStep
						iStep:=0; // Idle Step
					END_IF
		
				2: (* Start Z move *)
					GV_Axes.stAxisZ.lrAutoPosAbs:=stToolLocation.lrZcoord+lrToolDistance;
					GV_Axes.stAxisZ.bAutoCmdAbs:=TRUE;
					(*Log*)
						PRG_Log_WM.fbLogWM.M_Write_Log('FB_202_Action_PickPlaceToolMag : 2_AboveLocation : 2 : Start Z move');
					iSubStep:=3; // Next SubStep

				3: (* Wait Z move done *)
				   IF GV_Axes.stAxisZ.bAutoDone THEN
						GV_Axes.stAxisZ.bAutoCmdAbs:=FALSE;
						(*Log*)
							PRG_Log_WM.fbLogWM.M_Write_Log('FB_202_Action_PickPlaceToolMag : 2_AboveLocation : 3 : Z move done');
						iSubStep:=4; // Next SubStep
					ELSIF GV_Axes.stAxisZ.stDriveAx8206.AxisRef.Status.Error OR GV_Axes.stAxisZ.stDriveAx8206.AxisRef.Status.ErrorStop OR GV_Axes.stAxisZ.stDriveAx8206.AxisRef.Status.ErrorID<>0 THEN
						bError:=TRUE;
						udiErrorID:=231; // 211 = Step 2 SubStep 3 Error Axis Z 1
						GV_Axes.stAxisZ.bAutoCmdAbs:=FALSE;
						tonTimeoutMovex.IN:=FALSE;
						(*Log*)
							PRG_Log_WM.fbLogWM.M_Write_Log('FB_202_Action_PickPlaceToolMag : 2_AboveLocation=Error');
							PRG_Log_WM.fbLogWM.M_Write_Log(CONCAT('FB_202_Action_PickPlaceToolMag : ErrorID=',UDINT_TO_STRING(udiErrorID)));
						iSubStep:=0; // Stop SubStep
						iStep:=0; // Idle Step
					END_IF
					
				4: (* Start X move *)
					GV_Axes.stAxisX.lrAutoPosAbs:=stToolLocation.lrXcoord+lrOffsetX;
					GV_Axes.stAxisX.bAutoCmdAbs:=TRUE;
					(*Log*)
						PRG_Log_WM.fbLogWM.M_Write_Log('FB_202_Action_PickPlaceToolMag : 2_AboveLocation : 4 : Start X move');
					iSubStep:=5; // Next SubStep

				5: (* Wait X move done *)
				   IF GV_Axes.stAxisX.bAutoDone THEN
						GV_Axes.stAxisX.bAutoCmdAbs:=FALSE;
						(*Log*)
							PRG_Log_WM.fbLogWM.M_Write_Log('FB_202_Action_PickPlaceToolMag : 2_AboveLocation : 5 : X move done');
						iSubStep:=6; // Next SubStep
					ELSIF GV_Axes.stAxisX.stDriveAx8206.AxisRef.Status.Error OR GV_Axes.stAxisX.stDriveAx8206.AxisRef.Status.ErrorStop OR GV_Axes.stAxisX.stDriveAx8206.AxisRef.Status.ErrorID<>0 THEN
						bError:=TRUE;
						udiErrorID:=251; // 251 = Step 2 SubStep 5 Error Axis X 1
						GV_Axes.stAxisX.bAutoCmdAbs:=FALSE;
						tonTimeoutMovex.IN:=FALSE;
						(*Log*)
							PRG_Log_WM.fbLogWM.M_Write_Log('FB_202_Action_PickPlaceToolMag : 2_AboveLocation=Error');
							PRG_Log_WM.fbLogWM.M_Write_Log(CONCAT('FB_202_Action_PickPlaceToolMag : ErrorID=',UDINT_TO_STRING(udiErrorID)));
						iSubStep:=0; // Stop SubStep
						iStep:=0; // Idle Step
					END_IF

				6: (* Start Y move *)
					GV_Axes.stAxisY.lrAutoPosAbs:=stToolLocation.lrYcoord+lrOffsetY;
					GV_Axes.stAxisY.bAutoCmdAbs:=TRUE;
					(*Log*)
						PRG_Log_WM.fbLogWM.M_Write_Log('FB_202_Action_PickPlaceToolMag : 2_AboveLocation : 6 : Start Y move');
					iSubStep:=7; // Next Step

				7: (* Wait Y move done *)
				   IF GV_Axes.stAxisY.bAutoDone THEN
						GV_Axes.stAxisY.bAutoCmdAbs:=FALSE;
						tonTimeoutMovex.IN:=FALSE;
						(*Log*)
							PRG_Log_WM.fbLogWM.M_Write_Log('FB_202_Action_PickPlaceToolMag : 2_AboveLocation : 7 : Y move done');
							PRG_Log_WM.fbLogWM.M_Write_Log('FB_202_Action_PickPlaceToolMag : 2_AboveLocation->3_GripperUnclamp');
						iSubStep:=0; // End SubStep
						iStep:=3; // Next Step
					ELSIF GV_Axes.stAxisY.stDriveAx8206.AxisRef.Status.Error OR GV_Axes.stAxisY.stDriveAx8206.AxisRef.Status.ErrorStop OR GV_Axes.stAxisY.stDriveAx8206.AxisRef.Status.ErrorID<>0 THEN
						bError:=TRUE;
						udiErrorID:=271; // 271 = Step 2 SubStep 7 Error Axis Y 1
						GV_Axes.stAxisY.bAutoCmdAbs:=FALSE;
						tonTimeoutMovex.IN:=FALSE;
						(*Log*)
							PRG_Log_WM.fbLogWM.M_Write_Log('FB_202_Action_PickPlaceToolMag : 2_AboveLocation=Error');
							PRG_Log_WM.fbLogWM.M_Write_Log(CONCAT('FB_202_Action_PickPlaceToolMag : ErrorID=',UDINT_TO_STRING(udiErrorID)));
						iSubStep:=0; // Stop SubStep
						iStep:=0; // Idle Step
					END_IF
					
			END_CASE	
		
			IF tonTimeoutMovex.Q AND tonTimeoutMovex.PT<>T#0S THEN // Timeout 
				bError:=TRUE;
				udiErrorID:=299; // 299 = Step 2 Error Timeout 99
				GV_Axes.stAxisZ.bAutoCmdAbs:=FALSE;
				GV_Axes.stAxisX.bAutoCmdAbs:=FALSE;
				GV_Axes.stAxisY.bAutoCmdAbs:=FALSE;
				tonTimeoutMovex.IN:=FALSE;
				(*Log*)
					PRG_Log_WM.fbLogWM.M_Write_Log('FB_202_Action_PickPlaceToolMag : 2_AboveLocation=Error');
					PRG_Log_WM.fbLogWM.M_Write_Log(CONCAT('FB_202_Action_PickPlaceToolMag : ErrorID=',UDINT_TO_STRING(udiErrorID)));
				iSubStep:=0;
				iStep:=0;
			END_IF

		3: (* Step 3 = Operate manipulator gripper to unclamp *)
			eGripperMode:=ENUM_Gripper_Mode.Open; // Gripper mode
			tGripperTime:=tMouvementGripperOpen; // Gripper mouvement time
			bGripperSensor:=bCheckSensorGripperOpen; // Gripper check sensor
			
			IF (NOT fbGripper.bStart) AND (NOT fbGripper.bBusy) THEN // Gripper Start
				fbGripper.bStart:=TRUE;
			END_IF
			IF fbGripper.bDone THEN // Gripper Done
				fbGripper.bStart:=FALSE;
				(*Log*)
					PRG_Log_WM.fbLogWM.M_Write_Log('FB_202_Action_PickPlaceToolMag : 3_GripperUnclamp->4_Location');
				iSubStep:=0; // For next Step
				iStep:=4; // Next Step
			ELSIF fbGripper.bError THEN // Gripper Error
				bError:=TRUE;
				udiErrorID:=300+fbGripper.udiErrorID; // 3xx = Step 3 Error + Error xx fbGripper
				fbGripper.bStart:=FALSE;
				(*Log*)
					PRG_Log_WM.fbLogWM.M_Write_Log('FB_202_Action_PickPlaceToolMag : 3_GripperUnclamp=Error');
					PRG_Log_WM.fbLogWM.M_Write_Log(CONCAT('FB_202_Action_PickPlaceToolMag : ErrorID=',UDINT_TO_STRING(udiErrorID)));
				iStep:=0; // Idle Step
			END_IF

		4: (* Step 4 = Move the manipulator on the tool/location (Z-1mm) *)
			tonTimeoutMovex.PT:=tMovexTimeout;
			tonTimeoutMovex.IN:=TRUE;
			
			CASE iSubStep OF
        
				0: (* Start Z move *)
					GV_Axes.stAxisZ.lrAutoPosAbs:=stToolLocation.lrZcoord-1;
					GV_Axes.stAxisZ.bAutoCmdAbs:=TRUE;
					(*Log*)
						PRG_Log_WM.fbLogWM.M_Write_Log('FB_202_Action_PickPlaceToolMag : 4_Location : 0 : Start Z move home');
					iSubStep:=1; // Next SubStep

				1: (* Wait Z move done *)
				   IF GV_Axes.stAxisZ.bAutoDone THEN
						GV_Axes.stAxisZ.bAutoCmdAbs:=FALSE;
						tonTimeoutMovex.IN:=FALSE;
						(*Log*)
							PRG_Log_WM.fbLogWM.M_Write_Log('FB_202_Action_PickPlaceToolMag : 4_Location : 1 : Z move done');
							PRG_Log_WM.fbLogWM.M_Write_Log('FB_202_Action_PickPlaceToolMag : 4_Location->5_GripperClamp');
						iSubStep:=0; // End SubStep
						iStep:=5; // Next Step
					ELSIF GV_Axes.stAxisZ.stDriveAx8206.AxisRef.Status.Error OR GV_Axes.stAxisZ.stDriveAx8206.AxisRef.Status.ErrorStop OR GV_Axes.stAxisZ.stDriveAx8206.AxisRef.Status.ErrorID<>0 THEN
						bError:=TRUE;
						udiErrorID:=411; // 411 = Step 4 SubStep 1 Error Axis Z 1
						GV_Axes.stAxisZ.bAutoCmdAbs:=FALSE;
						tonTimeoutMovex.IN:=FALSE;
						(*Log*)
							PRG_Log_WM.fbLogWM.M_Write_Log('FB_202_Action_PickPlaceToolMag : 4_Location=Error');
							PRG_Log_WM.fbLogWM.M_Write_Log(CONCAT('FB_202_Action_PickPlaceToolMag : ErrorID=',UDINT_TO_STRING(udiErrorID)));
						iSubStep:=0; // Stop SubStep
						iStep:=0; // Idle Step
					END_IF
					
			END_CASE

			IF tonTimeoutMovex.Q AND tonTimeoutMovex.PT<>T#0S THEN // Timeout 
				bError:=TRUE;
				udiErrorID:=299; // 299 = Step 2 Error Timeout 99
				GV_Axes.stAxisZ.bAutoCmdAbs:=FALSE;
				GV_Axes.stAxisX.bAutoCmdAbs:=FALSE;
				GV_Axes.stAxisY.bAutoCmdAbs:=FALSE;
				tonTimeoutMovex.IN:=FALSE;
				(*Log*)
					PRG_Log_WM.fbLogWM.M_Write_Log('FB_202_Action_PickPlaceToolMag : 4_Location=Error');
					PRG_Log_WM.fbLogWM.M_Write_Log(CONCAT('FB_202_Action_PickPlaceToolMag : ErrorID=',UDINT_TO_STRING(udiErrorID)));
				iSubStep:=0;
				iStep:=0;
			END_IF

		5: (* Step 5 = Release manipulator gripper to clamp *)
			eGripperMode:=ENUM_Gripper_Mode.Close;
			tGripperTime:=tMouvementGripperClose; // Gripper mouvement time
			bGripperSensor:=bCheckSensorGripperClose; // Gripper check sensor
			
			IF (NOT fbGripper.bStart) AND (NOT fbGripper.bBusy) THEN // Gripper Start
				fbGripper.bStart:=TRUE;
			END_IF
			IF fbGripper.bDone THEN // Gripper Done
				fbGripper.bStart:=FALSE;
				(*Memory*)
					stToolLocation.bToolPresence:=FALSE; // Transfer Memory from Magazine to Manipulator
					GV_Tool_Magazine.stManipulator.iAbsLocationNumberMemory:=stToolLocation.iAbsLocationNumber; // Transfer Memory from Magazine to Manipulator
					GV_Tool_Magazine.stManipulator.iRelLocationNumberMemory:=stToolLocation.iRelLocationNumber; // Transfer Memory from Magazine to Manipulator
				(*Log*)
					PRG_Log_WM.fbLogWM.M_Write_Log('FB_202_Action_PickPlaceToolMag : 5_GripperClamp->6_FrontLocation');
				iSubStep:=0; // For next Step
				iStep:=6; // Next Step
			ELSIF fbGripper.bError THEN // Gripper Error
				bBusy:=FALSE;
				bError:=TRUE;
				udiErrorID:=500+fbGripper.udiErrorID; // 5xx = Step 5 Error + Error xx fbGripper
				fbGripper.bStart:=FALSE;
				(*Log*)
					PRG_Log_WM.fbLogWM.M_Write_Log('FB_202_Action_PickPlaceToolMag : 5_GripperClamp=Error');
					PRG_Log_WM.fbLogWM.M_Write_Log(CONCAT('FB_202_Action_PickPlaceToolMag : ErrorID=',UDINT_TO_STRING(udiErrorID)));
				iStep:=0; // Idle Step
			END_IF

		6: (* Step 6 = Move the manipulator in front of the tool/location (Z->Y0) -> Pick_Tool *)
			tonTimeoutMovex.PT:=tMovexTimeout;
			tonTimeoutMovex.IN:=TRUE;
			
			CASE iSubStep OF
        
				0: (* Start Z move *)
					GV_Axes.stAxisZ.lrAutoPosAbs:=stToolLocation.lrZcoord;
					GV_Axes.stAxisZ.bAutoCmdAbs:=TRUE;
					(*Log*)
						PRG_Log_WM.fbLogWM.M_Write_Log('FB_202_Action_PickPlaceToolMag : 6_FrontLocation : 0 : Start Z');
					iSubStep:=1; // Next SubStep

				1: (* Wait Z move done *)
				   IF GV_Axes.stAxisZ.bAutoDone THEN
						GV_Axes.stAxisZ.bAutoCmdAbs:=FALSE;
						(*Log*)
							PRG_Log_WM.fbLogWM.M_Write_Log('FB_202_Action_PickPlaceToolMag : 6_FrontLocation : 1 : Z move done');
						iSubStep:=2; // Next SubStep
					ELSIF GV_Axes.stAxisZ.stDriveAx8206.AxisRef.Status.Error OR GV_Axes.stAxisZ.stDriveAx8206.AxisRef.Status.ErrorStop OR GV_Axes.stAxisZ.stDriveAx8206.AxisRef.Status.ErrorID<>0 THEN
						bError:=TRUE;
						udiErrorID:=611; // 611 = Step 6 SubStep 1 Error Axis Z 1
						GV_Axes.stAxisZ.bAutoCmdAbs:=FALSE;
						tonTimeoutMovex.IN:=FALSE;
						(*Log*)
							PRG_Log_WM.fbLogWM.M_Write_Log('FB_202_Action_PickPlaceToolMag : 6_FrontLocation=Error');
							PRG_Log_WM.fbLogWM.M_Write_Log(CONCAT('FB_202_Action_PickPlaceToolMag : ErrorID=',UDINT_TO_STRING(udiErrorID)));
						iSubStep:=0; // Stop SubStep
						iStep:=0; // Idle Step
					END_IF

				2: (* Start Y move *)
					GV_Axes.stAxisY.lrAutoPosAbs:=0;//stToolLocation.lrYcoord+GV_Tool_Magazine.lrYOffsetFrontLocation;
					GV_Axes.stAxisY.bAutoCmdAbs:=TRUE;
					(*Log*)
						PRG_Log_WM.fbLogWM.M_Write_Log('FB_202_Action_PickPlaceToolMag : 6_FrontLocation : 2 : Start Y move');
					iSubStep:=3; // Next SubStep

				3: (* Wait Y move done *)
				   IF GV_Axes.stAxisY.bAutoDone THEN
						GV_Axes.stAxisY.bAutoCmdAbs:=FALSE;
						tonTimeoutMovex.IN:=FALSE;
						(*Log*)
							PRG_Log_WM.fbLogWM.M_Write_Log('FB_202_Action_PickPlaceToolMag : 6_FrontLocation : 3 : Y move done');
							PRG_Log_WM.fbLogWM.M_Write_Log('FB_202_Action_PickPlaceToolMag : 6_FrontLocation->7_Location');
						iSubStep:=0; // End SubStep
						iStep:=7; // Next Step
					ELSIF GV_Axes.stAxisY.stDriveAx8206.AxisRef.Status.Error OR GV_Axes.stAxisY.stDriveAx8206.AxisRef.Status.ErrorStop OR GV_Axes.stAxisY.stDriveAx8206.AxisRef.Status.ErrorID<>0 THEN
						bError:=TRUE;
						udiErrorID:=731; // 631 = Step 6 SubStep 3 Error Axis Y 1
						GV_Axes.stAxisY.bAutoCmdAbs:=FALSE;
						tonTimeoutMovex.IN:=FALSE;
						(*Log*)
							PRG_Log_WM.fbLogWM.M_Write_Log('FB_202_Action_PickPlaceToolMag : 6_FrontLocation=Error');
							PRG_Log_WM.fbLogWM.M_Write_Log(CONCAT('FB_202_Action_PickPlaceToolMag : ErrorID=',UDINT_TO_STRING(udiErrorID)));
						iSubStep:=0; // Stop SubStep
						iStep:=0; // Idle Step
					END_IF
					
			END_CASE	
		
			IF tonTimeoutMovex.Q AND tonTimeoutMovex.PT<>T#0S THEN // Timeout 
				bError:=TRUE;
				udiErrorID:=699; // 699 = Step 6 Error Timeout 99
				GV_Axes.stAxisY.bAutoCmdAbs:=FALSE;
				tonTimeoutMovex.IN := FALSE;
				(*Log*)
					PRG_Log_WM.fbLogWM.M_Write_Log('FB_202_Action_PickPlaceToolMag : 6_FrontLocation=Error');
					PRG_Log_WM.fbLogWM.M_Write_Log(CONCAT('FB_202_Action_PickPlaceToolMag : ErrorID=',UDINT_TO_STRING(udiErrorID)));
				iSubStep:=0;
				iStep:=0;
			END_IF

		7: (* Step 7 = Move the manipulator on the tool/location (Y) -> Place_Tool *)
			tonTimeoutMovex.PT:=tMovexTimeout;
			tonTimeoutMovex.IN:=TRUE;
			
			CASE iSubStep OF
		
				0: (* Start Y move *)
					GV_Axes.stAxisY.lrAutoPosAbs:=stToolLocation.lrYcoord+lrOffsetY;
					GV_Axes.stAxisY.bAutoCmdAbs:=TRUE;
					(*Log*)
						PRG_Log_WM.fbLogWM.M_Write_Log('FB_202_Action_PickPlaceToolMag : 7_Location : 0 : Start Y move');
					iSubStep:=1; // Next SubStep

				1: (* Wait Y move done *)
				   IF GV_Axes.stAxisY.bAutoDone THEN
						GV_Axes.stAxisY.bAutoCmdAbs:=FALSE;
						tonTimeoutMovex.IN:=FALSE;
						(*Log*)
							PRG_Log_WM.fbLogWM.M_Write_Log('FB_202_Action_PickPlaceToolMag : 7_Location : 1 : Y move done');
							PRG_Log_WM.fbLogWM.M_Write_Log('FB_202_Action_PickPlaceToolMag : 7_Location->8_GripperUnclamp');
						iSubStep:=0; // End SubStep
						iStep:=8; // Next Step
					ELSIF GV_Axes.stAxisY.stDriveAx8206.AxisRef.Status.Error OR GV_Axes.stAxisY.stDriveAx8206.AxisRef.Status.ErrorStop OR GV_Axes.stAxisY.stDriveAx8206.AxisRef.Status.ErrorID<>0 THEN
						bError:=TRUE;
						udiErrorID:=711; // 711 = Step 7 SubStep 1 Error Axis Y 1
						GV_Axes.stAxisY.bAutoCmdAbs:=FALSE;
						tonTimeoutMovex.IN:=FALSE;
						(*Log*)
							PRG_Log_WM.fbLogWM.M_Write_Log('FB_202_Action_PickPlaceToolMag : 7_Location=Error');
							PRG_Log_WM.fbLogWM.M_Write_Log(CONCAT('FB_202_Action_PickPlaceToolMag : ErrorID=',UDINT_TO_STRING(udiErrorID)));
						iSubStep:=0; // Stop SubStep
						iStep:=0; // Idle Step
					END_IF
					
			END_CASE	
		
			IF tonTimeoutMovex.Q AND tonTimeoutMovex.PT<>T#0S THEN // Timeout 
				bError:=TRUE;
				udiErrorID:=799; // 799 = Step 7 Error Timeout 99
				GV_Axes.stAxisY.bAutoCmdAbs:=FALSE;
				tonTimeoutMovex.IN := FALSE;
				(*Log*)
					PRG_Log_WM.fbLogWM.M_Write_Log('FB_202_Action_PickPlaceToolMag : 7_Location=Error');
					PRG_Log_WM.fbLogWM.M_Write_Log(CONCAT('FB_202_Action_PickPlaceToolMag : ErrorID=',UDINT_TO_STRING(udiErrorID)));
				iSubStep:=0;
				iStep:=0;
			END_IF

		8: (* Step 8 = Operate manipulator gripper to unclamp *)
			eGripperMode:=ENUM_Gripper_Mode.Open; // Gripper mode
			tGripperTime:=tMouvementGripperOpen; // Gripper mouvement time
			bGripperSensor:=bCheckSensorGripperOpen; // Gripper check sensor
			
			IF (NOT fbGripper.bStart) AND (NOT fbGripper.bBusy) THEN // Gripper Start
				fbGripper.bStart:=TRUE;
			END_IF
			IF fbGripper.bDone THEN // Gripper Done
				fbGripper.bStart:=FALSE;
				(*Memory*)
					stToolLocation.bToolPresence:=TRUE; // Transfer Memory from Manipulator to Magazine
					GV_Tool_Magazine.stManipulator.iAbsLocationNumberMemory:=0; // Reset Manipulator Memory
					GV_Tool_Magazine.stManipulator.iRelLocationNumberMemory:=0; // Reset Manipulator Memory
				(*Log*)
					PRG_Log_WM.fbLogWM.M_Write_Log('FB_202_Action_PickPlaceToolMag : 8_GripperUnclamp->9_AbovetLocation');
				iSubStep:=0; // For next Step
				iStep:=9; // Next Step
			ELSIF fbGripper.bError THEN // Gripper Error
				bError:=TRUE;
				udiErrorID:=800+fbGripper.udiErrorID; // 3xx = Step 8 Error + Error xx fbGripper
				fbGripper.bStart:=FALSE;
				(*Log*)
					PRG_Log_WM.fbLogWM.M_Write_Log('FB_202_Action_PickPlaceToolMag : 8_GripperUnclamp=Error');
					PRG_Log_WM.fbLogWM.M_Write_Log(CONCAT('FB_202_Action_PickPlaceToolMag : ErrorID=',UDINT_TO_STRING(udiErrorID)));
				iStep:=0; // Idle Step
			END_IF

		9: (* Step 9 = Move the manipulator above the tool/location (Zoffset) *)
			tonTimeoutMovex.PT:=tMovexTimeout;
			tonTimeoutMovex.IN:=TRUE;
		
			CASE iSubStep OF
		
				0: (* Start Z move *)
					GV_Axes.stAxisZ.lrAutoPosAbs:=stToolLocation.lrZcoord+lrToolDistance;
					GV_Axes.stAxisZ.bAutoCmdAbs:=TRUE;
					(*Log*)
						PRG_Log_WM.fbLogWM.M_Write_Log('FB_202_Action_PickPlaceToolMag : 9_AbovetLocation : 0 : Start Z');
					iSubStep:=1; // Next SubStep

				1: (* Wait Z move done *)
				   IF GV_Axes.stAxisZ.bAutoDone THEN
						GV_Axes.stAxisZ.bAutoCmdAbs:=FALSE;
						(*Log*)
							PRG_Log_WM.fbLogWM.M_Write_Log('FB_202_Action_PickPlaceToolMag : 9_AbovetLocation : 1 : Z move done');
							PRG_Log_WM.fbLogWM.M_Write_Log('FB_202_Action_PickPlaceToolMag : 9_AbovetLocation->10_GripperClamp');
						iSubStep:=0; // Next SubStep
						iStep:=10; // Next Step
					ELSIF GV_Axes.stAxisZ.stDriveAx8206.AxisRef.Status.Error OR GV_Axes.stAxisZ.stDriveAx8206.AxisRef.Status.ErrorStop OR GV_Axes.stAxisZ.stDriveAx8206.AxisRef.Status.ErrorID<>0 THEN
						bError:=TRUE;
						udiErrorID:=911; // 911 = Step 9 SubStep 1 Error Axis Z 1
						GV_Axes.stAxisZ.bAutoCmdAbs:=FALSE;
						tonTimeoutMovex.IN:=FALSE;
						(*Log*)
							PRG_Log_WM.fbLogWM.M_Write_Log('FB_202_Action_PickPlaceToolMag : 9_AbovetLocation=Error');
							PRG_Log_WM.fbLogWM.M_Write_Log(CONCAT('FB_202_Action_PickPlaceToolMag : ErrorID=',UDINT_TO_STRING(udiErrorID)));
						iSubStep:=0; // Stop SubStep
						iStep:=0; // Idle Step
					END_IF

			END_CASE
				
			IF tonTimeoutMovex.Q AND tonTimeoutMovex.PT<>T#0S THEN // Timeout 
				bError:=TRUE;
				udiErrorID:=999; // 999 = Step 9 Error Timeout 99
				GV_Axes.stAxisY.bAutoCmdAbs:=FALSE;
				tonTimeoutMovex.IN := FALSE;
				(*Log*)
					PRG_Log_WM.fbLogWM.M_Write_Log('FB_202_Action_PickPlaceToolMag : 9_AbovetLocation=Error');
					PRG_Log_WM.fbLogWM.M_Write_Log(CONCAT('FB_202_Action_PickPlaceToolMag : ErrorID=',UDINT_TO_STRING(udiErrorID)));
				iSubStep:=0;
				iStep:=0;
			END_IF
		
		10: (* Step 10 = Release manipulator gripper to clamp *)
			eGripperMode:=ENUM_Gripper_Mode.Close;
			tGripperTime:=tMouvementGripperClose; // Gripper mouvement time
			bGripperSensor:=bCheckSensorGripperClose; // Gripper check sensor
			
			IF (NOT fbGripper.bStart) AND (NOT fbGripper.bBusy) THEN // Gripper Start
				fbGripper.bStart:=TRUE;
			END_IF
			IF fbGripper.bDone THEN // Gripper Done
				fbGripper.bStart:=FALSE;
				(*Memory*)
					//stToolLocation.bToolPresence:=FALSE; // Transfer Memory from Magazine to Manipulator
					//GV_Tool_Magazine.stManipulator.iAbsLocationNumberMemory:=stToolLocation.iAbsLocationNumber; // Transfer Memory from Magazine to Manipulator
					//GV_Tool_Magazine.stManipulator.iRelLocationNumberMemory:=stToolLocation.iRelLocationNumber; // Transfer Memory from Magazine to Manipulator
				(*Log*)
					PRG_Log_WM.fbLogWM.M_Write_Log('FB_202_Action_PickPlaceToolMag : 10_GripperClamp->11_FrontLocation');
				iSubStep:=0; // For next Step
				iStep:=11; // Next Step
			ELSIF fbGripper.bError THEN // Gripper Error
				bBusy:=FALSE;
				bError:=TRUE;
				udiErrorID:=500+fbGripper.udiErrorID; // 5xx = Step 5 Error + Error xx fbGripper
				fbGripper.bStart:=FALSE;
				(*Log*)
					PRG_Log_WM.fbLogWM.M_Write_Log('FB_202_Action_PickPlaceToolMag : 10_GripperClamp=Error');
					PRG_Log_WM.fbLogWM.M_Write_Log(CONCAT('FB_202_Action_PickPlaceToolMag : ErrorID=',UDINT_TO_STRING(udiErrorID)));
				iStep:=0; // Idle Step
			END_IF
		
		11 : (* Step 11 = Move the manipulator in front of the tool/location (Y0) *)
			tonTimeoutMovex.PT:=tMovexTimeout;
			tonTimeoutMovex.IN:=TRUE;
		
			CASE iSubStep OF
		
				0: (* Start Y move *)
					GV_Axes.stAxisY.lrAutoPosAbs:=0;//stToolLocation.lrYcoord+GV_Tool_Magazine.lrYOffsetFrontLocation;
					GV_Axes.stAxisY.bAutoCmdAbs:=TRUE;
					(*Log*)
						PRG_Log_WM.fbLogWM.M_Write_Log('FB_202_Action_PickPlaceToolMag : 11_FrontLocation : 0 : Start Y move');
					iSubStep:=1; // Next SubStep

				1: (* Wait Y move done *)
				   IF GV_Axes.stAxisY.bAutoDone THEN
						GV_Axes.stAxisY.bAutoCmdAbs:=FALSE;
						tonTimeoutMovex.IN:=FALSE;
						(*Log*)
							PRG_Log_WM.fbLogWM.M_Write_Log('FB_202_Action_PickPlaceToolMag : 11_FrontLocation : 1 : Y move done');
							PRG_Log_WM.fbLogWM.M_Write_Log('FB_202_Action_PickPlaceToolMag : 11_FrontLocation->0_Idle');
						iSubStep:=0; // End SubStep
						iStep:=0; // End Step
						bDone:=TRUE;
						bBusy:=FALSE;
					ELSIF GV_Axes.stAxisY.stDriveAx8206.AxisRef.Status.Error OR GV_Axes.stAxisY.stDriveAx8206.AxisRef.Status.ErrorStop OR GV_Axes.stAxisY.stDriveAx8206.AxisRef.Status.ErrorID<>0 THEN
						bError:=TRUE;
						udiErrorID:=931; // 711 = Step 9 SubStep 3 Error Axis Y 1
						GV_Axes.stAxisY.bAutoCmdAbs:=FALSE;
						tonTimeoutMovex.IN:=FALSE;
						(*Log*)
							PRG_Log_WM.fbLogWM.M_Write_Log('FB_202_Action_PickPlaceToolMag : 11_FrontLocation=Error');
							PRG_Log_WM.fbLogWM.M_Write_Log(CONCAT('FB_202_Action_PickPlaceToolMag : ErrorID=',UDINT_TO_STRING(udiErrorID)));
						iSubStep:=0; // Stop SubStep
						iStep:=0; // Idle Step
					END_IF
			END_CASE
				
			IF tonTimeoutMovex.Q AND tonTimeoutMovex.PT<>T#0S THEN // Timeout 
				bError:=TRUE;
				udiErrorID:=999; // 999 = Step 9 Error Timeout 99
				GV_Axes.stAxisY.bAutoCmdAbs:=FALSE;
				tonTimeoutMovex.IN := FALSE;
				(*Log*)
					PRG_Log_WM.fbLogWM.M_Write_Log('FB_202_Action_PickPlaceToolMag : 11_FrontLocation=Error');
					PRG_Log_WM.fbLogWM.M_Write_Log(CONCAT('FB_202_Action_PickPlaceToolMag : ErrorID=',UDINT_TO_STRING(udiErrorID)));
				iSubStep:=0;
				iStep:=0;
			END_IF
			
	END_CASE

END_FUNCTION_BLOCK

// ---- 09_Tool_Magazine/03_POUs/01_PRGs/PRG_Tool_Magazine_Type1_Refresh.TcPOU
PROGRAM PRG_Tool_Magazine_Type1_Refresh
VAR
	(** INT **)
	iRackLoop : INT := 0 ; // Use in a FOR Loop
	iLocationLoop : INT := 0 ; // Use in a FOR Loop
END_VAR

//-----------------------------------------------------------------------------------------
//
//                  		PRG_Tool_Magazine_Type1_Refresh
//
//				Paramétrage magasin d'outils sur demande ou toute 1ère fois 	
//			ATTENTION -> REINITIALISE LES COORDONEES DES EMPLACEMENTS DU MAGASIN !!!	
//-----------------------------------------------------------------------------------------
//
//Auteur: G.GOETZ
//Création: 14.01.2026
//Dernière modification : 19.03.2026 (G.GOETZ)
//       			
//-----------------------------------------------------------------------------------------
//
//     							Liste des modifications  	
//
// 14.01.2026 (G.GOETZ) -> Création		
// 19.03.2026 (G.GOETZ) -> X,Y,Z lrCoord... Calcul
//-----------------------------------------------------------------------------------------

(** SETUP PROCESS **)
	GV_Tool_Magazine.lrYOffsetFrontLocation:=GV_HMI.stMagazineSettings.lrYOffsetFrontLocation; // MIN = ? = GV_Tool_Magazine.lrMinYOffsetFrontLocation // MAX = ? = GV_Tool_Magazine.lrMaxYOffsetFrontLocation // -> from HMI screen : Magazine Settings
	GV_Tool_Magazine.lrYOffsetFrontLocation:=GV_HMI.stMagazineSettings.lrZOffsetAboveLocation; // MIN = ? = GV_Tool_Magazine.lrMinZOffsetAboveLocation // MAX = ? = GV_Tool_Magazine.lrMaxZOffsetAboveLocation // -> from HMI screen : Magazine Settings
	GV_Tool_Magazine.lrZOffsetAboveArmGripper1:=GV_HMI.stMagazineSettings.lrZOffsetAboveArmGripper1; // MIN = ? = GV_Tool_Magazine.lrZOffsetAboveArmGripper1 // MAX = ? = GV_Tool_Magazine.lrMaxZOffsetAboveArmGripper1 // -> from HMI screen : Magazine Settings
	GV_Tool_Magazine.lrZOffsetAboveArmGripper2:=GV_HMI.stMagazineSettings.lrZOffsetAboveArmGripper2; // MIN = ? = GV_Tool_Magazine.lrZOffsetAboveArmGripper2 // MAX = ? = GV_Tool_Magazine.lrMaxZOffsetAboveArmGripper2 // -> from HMI screen : Magazine Settings
	(* Limit *)
		(*Limit Y Front Location*) // Not used
			IF GV_Tool_Magazine.lrYOffsetFrontLocation<GV_Tool_Magazine.lrMinYOffsetFrontLocation THEN
				GV_Tool_Magazine.lrYOffsetFrontLocation:=GV_Tool_Magazine.lrMinYOffsetFrontLocation;
			END_IF
			IF GV_Tool_Magazine.lrYOffsetFrontLocation>GV_Tool_Magazine.lrMaxYOffsetFrontLocation THEN
				GV_Tool_Magazine.lrYOffsetFrontLocation:=GV_Tool_Magazine.lrMaxYOffsetFrontLocation;
			END_IF
		(*Limit Z Above Location*)
			IF GV_Tool_Magazine.lrZOffsetAboveLocation<GV_Tool_Magazine.lrMinZOffsetAboveLocation THEN
				GV_Tool_Magazine.lrZOffsetAboveLocation:=GV_Tool_Magazine.lrMinZOffsetAboveLocation;
			END_IF
			IF GV_Tool_Magazine.lrZOffsetAboveLocation>GV_Tool_Magazine.lrMaxZOffsetAboveLocation THEN
				GV_Tool_Magazine.lrZOffsetAboveLocation:=GV_Tool_Magazine.lrMaxZOffsetAboveLocation;
			END_IF
		(*Limit Z Above ArmGripper1*)
			IF GV_Tool_Magazine.lrZOffsetAboveArmGripper1<GV_Tool_Magazine.lrMinZOffsetAboveArmGripper1 THEN
				GV_Tool_Magazine.lrZOffsetAboveArmGripper1:=GV_Tool_Magazine.lrMinZOffsetAboveArmGripper1;
			END_IF
			IF GV_Tool_Magazine.lrZOffsetAboveArmGripper1>GV_Tool_Magazine.lrMaxZOffsetAboveArmGripper1 THEN
				GV_Tool_Magazine.lrZOffsetAboveArmGripper1:=GV_Tool_Magazine.lrMaxZOffsetAboveArmGripper1;
			END_IF
		(*Limit Z Above ArmGripper2*)
			IF GV_Tool_Magazine.lrZOffsetAboveArmGripper2<GV_Tool_Magazine.lrMinZOffsetAboveArmGripper2 THEN
				GV_Tool_Magazine.lrZOffsetAboveArmGripper2:=GV_Tool_Magazine.lrMinZOffsetAboveArmGripper2;
			END_IF
			IF GV_Tool_Magazine.lrZOffsetAboveArmGripper2>GV_Tool_Magazine.lrMaxZOffsetAboveArmGripper2 THEN
				GV_Tool_Magazine.lrZOffsetAboveArmGripper2:=GV_Tool_Magazine.lrMaxZOffsetAboveArmGripper2;
			END_IF
		
(** SETUP RACK **)
	GV_Tool_Magazine.iMaxRelRackTop:=GV_HMI.stMagazineSettings.iMaxRelRackTop; // MAX = 5 = GV_Tool_Magazine.iMaxAbsRackTop // -> from HMI screen : Magazine Settings
	GV_Tool_Magazine.iMaxRelRackBottom:=GV_HMI.stMagazineSettings.iMaxRelRackBottom; // MAX = 3 = GV_Tool_Magazine.iMaxAbsRackBottom // -> from HMI screen : Magazine Settings
	(* Limit *)
		(*Limit Rack Top*)
			IF GV_Tool_Magazine.iMaxRelRackTop<0 THEN
				GV_Tool_Magazine.iMaxRelRackTop:=0;
			END_IF
			IF GV_Tool_Magazine.iMaxRelRackTop>GV_Tool_Magazine.iMaxAbsRackTop THEN
				GV_Tool_Magazine.iMaxRelRackTop:=GV_Tool_Magazine.iMaxAbsRackTop;
			END_IF
		(*Limit Rack Bottom*)
			IF GV_Tool_Magazine.iMaxRelRackBottom<0 THEN
				GV_Tool_Magazine.iMaxRelRackBottom:=0;
			END_IF
			IF GV_Tool_Magazine.iMaxRelRackBottom>GV_Tool_Magazine.iMaxAbsRackBottom THEN
				GV_Tool_Magazine.iMaxRelRackBottom:=GV_Tool_Magazine.iMaxAbsRackBottom;
			END_IF	
		(*Limit Rack*)
			IF GV_Tool_Magazine.iMaxRelRack<0 THEN
				GV_Tool_Magazine.iMaxRelRack:=0;
			END_IF
			IF GV_Tool_Magazine.iMaxRelRack>GV_Tool_Magazine.iMaxAbsRack THEN
				GV_Tool_Magazine.iMaxRelRack:=GV_Tool_Magazine.iMaxAbsRack;
			END_IF
	GV_Tool_Magazine.iMaxRelRack:=GV_Tool_Magazine.iMaxRelRackTop+GV_Tool_Magazine.iMaxRelRackBottom; // MAX = 5+3 = 8 = GV_Tool_Magazine.iMaxAbsRackTop+GV_Tool_Magazine.iMaxAbsRackBottom = GV_Tool_Magazine.iMaxAbsRack
	
	GV_Tool_Magazine.lrZLowestRackTop:=GV_HMI.stMagazineSettings.lrZLowestRackTop; // MIN = ? = GV_Tool_Magazine.lrMinZLowestRackTop // MAX = ? = GV_Tool_Magazine.lrMaxZLowestRackTop // -> from HMI screen : Magazine Settings
	GV_Tool_Magazine.lrZLowestRackBottom:=GV_HMI.stMagazineSettings.lrZLowestRackBottom; // MIN = ? = GV_Tool_Magazine.lrMinZLowestRackBottom // MAX = ? = GV_Tool_Magazine.lrMaxZLowestRackBottom // -> from HMI screen : Magazine Settings
	(* Limit *)
		(*Limit Z Lowest Rack Top*)
			IF GV_Tool_Magazine.lrZLowestRackTop<GV_Tool_Magazine.lrMinZLowestRackTop THEN
				GV_Tool_Magazine.lrZLowestRackTop:=GV_Tool_Magazine.lrMinZLowestRackTop;
			END_IF
			IF GV_Tool_Magazine.lrZLowestRackTop>GV_Tool_Magazine.lrMaxZLowestRackTop THEN
				GV_Tool_Magazine.lrZLowestRackTop:=GV_Tool_Magazine.lrMaxZLowestRackTop;
			END_IF
		(*Limit Z Lowest Rack Bottom*)
			IF GV_Tool_Magazine.lrZLowestRackBottom<GV_Tool_Magazine.lrMinZLowestRackBottom THEN
				GV_Tool_Magazine.lrZLowestRackBottom:=GV_Tool_Magazine.lrMinZLowestRackBottom;
			END_IF
			IF GV_Tool_Magazine.lrZLowestRackBottom>GV_Tool_Magazine.lrMaxZLowestRackBottom THEN
				GV_Tool_Magazine.lrZLowestRackBottom:=GV_Tool_Magazine.lrMaxZLowestRackBottom;
			END_IF
			
(** SETUP LOCATIONS IN RACK **)
	GV_Tool_Magazine.iMaxRelRackLocationTop:=GV_HMI.stMagazineSettings.iMaxRelRackLocationTop; // MAX = 19 = GV_Tool_Magazine.iMaxAbsLocationRackTop // -> from HMI screen : Magazine Settings
	GV_Tool_Magazine.iMaxRelRackLocationBottom:=GV_HMI.stMagazineSettings.iMaxRelRackLocationBottom; // MAX = 15 = GV_Tool_Magazine.iMaxAbsLocationRackBottom // -> from HMI screen : Magazine Settings
	(* Limit *)
		(*Limit Location in Rack Top*)
			IF GV_Tool_Magazine.iMaxRelRackLocationTop<0 THEN
				GV_Tool_Magazine.iMaxRelRackLocationTop:=0;
			END_IF
			IF GV_Tool_Magazine.iMaxRelRackLocationTop>GV_Tool_Magazine.iMaxAbsLocationRackTop THEN
				GV_Tool_Magazine.iMaxRelRackLocationTop:=GV_Tool_Magazine.iMaxAbsLocationRackTop;
			END_IF
		(*Limit Location in Rack Bottom*)
			IF GV_Tool_Magazine.iMaxRelRackLocationBottom<0 THEN
				GV_Tool_Magazine.iMaxRelRackLocationBottom:=0;
			END_IF
			IF GV_Tool_Magazine.iMaxRelRackLocationBottom>GV_Tool_Magazine.iMaxAbsLocationRackBottom THEN
				GV_Tool_Magazine.iMaxRelRackLocationBottom:=GV_Tool_Magazine.iMaxAbsLocationRackBottom;
			END_IF
	GV_Tool_Magazine.lrXLocationOffsetTop:=GV_HMI.stMagazineSettings.lrXLocationOffsetTop; // MIN = ? = GV_Tool_Magazine.lrMinXLocationOffsetTop // MAX = ? = GV_Tool_Magazine.lrMaxXLocationOffsetTop // -> from HMI screen : Magazine Settings
	GV_Tool_Magazine.lrYLocationOffsetTop:=GV_HMI.stMagazineSettings.lrYLocationOffsetTop; // MIN = ? = GV_Tool_Magazine.lrMinYLocationOffsetTop // MAX = ? = GV_Tool_Magazine.lrMaxYLocationOffsetTop // -> from HMI screen : Magazine Settings
	GV_Tool_Magazine.lrZLocationOffsetTop:=GV_HMI.stMagazineSettings.lrZLocationOffsetTop; // MIN = ? = GV_Tool_Magazine.lrMinZLocationOffsetTop // MAX = ? = GV_Tool_Magazine.lrMaxZLocationOffsetTop // -> from HMI screen : Magazine Settings
	GV_Tool_Magazine.lrXLocationOffsetBottom:=GV_HMI.stMagazineSettings.lrXLocationOffsetBottom; // MIN = ? = GV_Tool_Magazine.lrMinXLocationOffsetBottom // MAX = ? = GV_Tool_Magazine.lrMaxXLocationOffsetBottom // -> from HMI screen : Magazine Settings
	GV_Tool_Magazine.lrYLocationOffsetBottom:=GV_HMI.stMagazineSettings.lrYLocationOffsetBottom; // MIN = ? = GV_Tool_Magazine.lrMinYLocationOffsetBottom // MAX = ? = GV_Tool_Magazine.lrMaxYLocationOffsetBottom // -> from HMI screen : Magazine Settings
	GV_Tool_Magazine.lrZLocationOffsetBottom:=GV_HMI.stMagazineSettings.lrZLocationOffsetBottom; // MIN = ? = GV_Tool_Magazine.lrMinZLocationOffsetBottom // MAX = ? = GV_Tool_Magazine.lrMaxZLocationOffsetBottom // -> from HMI screen : Magazine Settings
	(* Limit *)
		(*Limit Offset X between Location at the Top*)
			IF GV_Tool_Magazine.lrXLocationOffsetTop<GV_Tool_Magazine.lrMinXLocationOffsetTop THEN
				GV_Tool_Magazine.lrXLocationOffsetTop:=GV_Tool_Magazine.lrMinXLocationOffsetTop;
			END_IF
			IF GV_Tool_Magazine.lrXLocationOffsetTop>GV_Tool_Magazine.lrMaxXLocationOffsetTop THEN
				GV_Tool_Magazine.lrXLocationOffsetTop:=GV_Tool_Magazine.lrMaxXLocationOffsetTop;
			END_IF
		(*Limit Offset Y between Location at the Top*)
			IF GV_Tool_Magazine.lrYLocationOffsetTop<GV_Tool_Magazine.lrMinYLocationOffsetTop THEN
				GV_Tool_Magazine.lrYLocationOffsetTop:=GV_Tool_Magazine.lrMinYLocationOffsetTop;
			END_IF
			IF GV_Tool_Magazine.lrYLocationOffsetTop>GV_Tool_Magazine.lrMaxYLocationOffsetTop THEN
				GV_Tool_Magazine.lrYLocationOffsetTop:=GV_Tool_Magazine.lrMaxYLocationOffsetTop;
			END_IF
		(*Limit Offset Z between Location at the Top*)
			IF GV_Tool_Magazine.lrZLocationOffsetTop<GV_Tool_Magazine.lrMinZLocationOffsetTop THEN
				GV_Tool_Magazine.lrZLocationOffsetTop:=GV_Tool_Magazine.lrMinZLocationOffsetTop;
			END_IF
			IF GV_Tool_Magazine.lrZLocationOffsetTop>GV_Tool_Magazine.lrMaxZLocationOffsetTop THEN
				GV_Tool_Magazine.lrZLocationOffsetTop:=GV_Tool_Magazine.lrMaxZLocationOffsetTop;
			END_IF
		(*Limit Offset X between Location at the Bottom*)
			IF GV_Tool_Magazine.lrXLocationOffsetBottom<GV_Tool_Magazine.lrMinXLocationOffsetBottom THEN
				GV_Tool_Magazine.lrXLocationOffsetBottom:=GV_Tool_Magazine.lrMinXLocationOffsetBottom;
			END_IF
			IF GV_Tool_Magazine.lrXLocationOffsetBottom>GV_Tool_Magazine.lrMaxXLocationOffsetBottom THEN
				GV_Tool_Magazine.lrXLocationOffsetBottom:=GV_Tool_Magazine.lrMaxXLocationOffsetBottom;
			END_IF
		(*Limit Offset Y between Location at the Bottom*)
			IF GV_Tool_Magazine.lrYLocationOffsetBottom<GV_Tool_Magazine.lrMinYLocationOffsetBottom THEN
				GV_Tool_Magazine.lrYLocationOffsetBottom:=GV_Tool_Magazine.lrMinYLocationOffsetBottom;
			END_IF
			IF GV_Tool_Magazine.lrYLocationOffsetBottom>GV_Tool_Magazine.lrMaxYLocationOffsetBottom THEN
				GV_Tool_Magazine.lrYLocationOffsetBottom:=GV_Tool_Magazine.lrMaxYLocationOffsetBottom;
			END_IF
		(*Limit Offset Z between Location at the Bottom*)
			IF GV_Tool_Magazine.lrZLocationOffsetBottom<GV_Tool_Magazine.lrMinZLocationOffsetBottom THEN
				GV_Tool_Magazine.lrZLocationOffsetBottom:=GV_Tool_Magazine.lrMinZLocationOffsetBottom;
			END_IF
			IF GV_Tool_Magazine.lrZLocationOffsetBottom>GV_Tool_Magazine.lrMaxZLocationOffsetBottom THEN
				GV_Tool_Magazine.lrZLocationOffsetBottom:=GV_Tool_Magazine.lrMaxZLocationOffsetBottom;
			END_IF
			
(** SETUP LOCATIONS **)
	GV_Tool_Magazine.iMaxRelLocationTop:=GV_Tool_Magazine.iMaxRelRackTop*GV_Tool_Magazine.iMaxRelRackLocationTop; // MAX = 5*19 = 95 = GV_Tool_Magazine.iMaxAbsRackTop*GV_Tool_Magazine.iMaxAbsRackLocationTop = GV_Tool_Magazine.iMaxAbsLocationTop
	GV_Tool_Magazine.iMaxRelLocationBottom:=GV_Tool_Magazine.iMaxRelRackBottom*GV_Tool_Magazine.iMaxRelRackLocationBottom; // MAX = 3*15 = 45 = GV_Tool_Magazine.iMaxAbsRackBottom*GV_Tool_Magazine.iMaxAbsRackLocationBottom = GV_Tool_Magazine.iMaxAbsLocationBottom
	GV_Tool_Magazine.iMaxRelLocation:=GV_Tool_Magazine.iMaxRelLocationTop+GV_Tool_Magazine.iMaxRelLocationBottom; // MAX  = 95+45 = 140 = GV_Tool_Magazine.iMaxAbsLocationTop+GV_Tool_Magazine.iMaxAbsLocationBottom = GV_Tool_Magazine.iMaxAbsLocation
	
	GV_Tool_Magazine.lrZAbsCompensationLocationTop:=0;//GV_HMI.stMagazineSettings.lrZAbsCompensationLocationTop; // mm // MAX = 10 = GV_Tool_Magazine.lrMaxAbsCompensationLocationTop  // -> from HMI screen : Magazine Settings
	GV_Tool_Magazine.lrZAbsCompensationLocationBottom:=0;//GV_HMI.stMagazineSettings.lrZAbsCompensationLocationBottom; // mm // MAX = 10 = GV_Tool_Magazine.lrMaxAbsCompensationLocationBottom // -> from HMI screen : Magazine Settings
	(* Limit *)		
		(*Limit Compensation Location Top*)
			IF GV_Tool_Magazine.lrZAbsCompensationLocationTop<GV_Tool_Magazine.lrMinAbsCompensationLocationTop THEN
				GV_Tool_Magazine.lrZAbsCompensationLocationTop:=GV_Tool_Magazine.lrMinAbsCompensationLocationTop;
			END_IF
			IF GV_Tool_Magazine.lrZAbsCompensationLocationTop>GV_Tool_Magazine.lrMaxAbsCompensationLocationTop THEN
				 GV_Tool_Magazine.lrZAbsCompensationLocationTop:=GV_Tool_Magazine.lrMaxAbsCompensationLocationTop;
			END_IF
		(*Limit Compensation Location Bottom*)
			IF GV_Tool_Magazine.lrZAbsCompensationLocationBottom<GV_Tool_Magazine.lrMinAbsCompensationLocationBottom THEN
				GV_Tool_Magazine.lrZAbsCompensationLocationBottom:=GV_Tool_Magazine.lrMinAbsCompensationLocationBottom;
			END_IF
			IF GV_Tool_Magazine.lrZAbsCompensationLocationBottom>GV_Tool_Magazine.lrMaxAbsCompensationLocationBottom THEN
				 GV_Tool_Magazine.lrZAbsCompensationLocationBottom:=GV_Tool_Magazine.lrMaxAbsCompensationLocationBottom;
			END_IF
	IF GV_Tool_Magazine.iMaxRelRackLocationTop>1 THEN
		GV_Tool_Magazine.lrZRelCompensationLocationTop:=GV_Tool_Magazine.lrZAbsCompensationLocationTop/(GV_Tool_Magazine.iMaxRelRackLocationTop-1);
		GV_Tool_Magazine.lrZRelCompensationLocationTop:=LINT_TO_LREAL(LREAL_TO_LINT(GV_Tool_Magazine.lrZRelCompensationLocationTop*1000.0))/1000.0; // Round 10e-3
	ELSE
		GV_Tool_Magazine.lrZRelCompensationLocationTop:=0;
	END_IF
	IF GV_Tool_Magazine.iMaxRelRackLocationBottom>1 THEN
		GV_Tool_Magazine.lrZRelCompensationLocationBottom:=GV_Tool_Magazine.lrZAbsCompensationLocationBottom/(GV_Tool_Magazine.iMaxRelRackLocationBottom-1);
		GV_Tool_Magazine.lrZRelCompensationLocationBottom:=LINT_TO_LREAL(LREAL_TO_LINT(GV_Tool_Magazine.lrZRelCompensationLocationBottom*1000.0))/1000.0; // Round 10e-3
	ELSE
		GV_Tool_Magazine.lrZRelCompensationLocationBottom:=0;
	END_IF	
		GV_Tool_Magazine.lrXFirstLocationTop:=GV_HMI.stMagazineSettings.lrXFirstLocationTop; // MIN = ? = GV_Tool_Magazine.lrMinXFirstLocationTop // MAX = ? = GV_Tool_Magazine.lrMaxXFirstLocationTop // -> from HMI screen : Magazine Settings
		GV_Tool_Magazine.lrXFirstLocationBottom:=GV_HMI.stMagazineSettings.lrXFirstLocationBottom; // MIN = ? = GV_Tool_Magazine.lrMinXFirstLocationBottom // MAX = ? = GV_Tool_Magazine.lrMaxXFirstLocationBottom // -> from HMI screen : Magazine Settings
		GV_Tool_Magazine.lrYLocationTop:=GV_HMI.stMagazineSettings.lrYLocationTop; // MIN = ? = GV_Tool_Magazine.lrMinYLocationTop // MAX = ? = GV_Tool_Magazine.lrMaxYLocationTop // -> from HMI screen : Magazine Settings
		GV_Tool_Magazine.lrYLocationBottom:=GV_HMI.stMagazineSettings.lrYLocationBottom; // MIN = ? = GV_Tool_Magazine.lrMinYLocationTop // MAX = ? = GV_Tool_Magazine.lrMaxYLocationTop // -> from HMI screen : Magazine Settings
	(* Limit *)
		(*Limit X First Location Top*)
			IF GV_Tool_Magazine.lrXFirstLocationTop<GV_Tool_Magazine.lrMinXFirstLocationTop THEN
				GV_Tool_Magazine.lrXFirstLocationTop:=GV_Tool_Magazine.lrMinXFirstLocationTop;
			END_IF
			IF GV_Tool_Magazine.lrXFirstLocationTop>GV_Tool_Magazine.lrMaxXFirstLocationTop THEN
				GV_Tool_Magazine.lrXFirstLocationTop:=GV_Tool_Magazine.lrMaxXFirstLocationTop;
			END_IF
		(*Limit X First Location Bottom*)
			IF GV_Tool_Magazine.lrXFirstLocationBottom<GV_Tool_Magazine.lrMinXFirstLocationBottom THEN
				GV_Tool_Magazine.lrXFirstLocationBottom:=GV_Tool_Magazine.lrMinXFirstLocationBottom;
			END_IF
			IF GV_Tool_Magazine.lrXFirstLocationBottom>GV_Tool_Magazine.lrMaxXFirstLocationBottom THEN
				GV_Tool_Magazine.lrXFirstLocationBottom:=GV_Tool_Magazine.lrMaxXFirstLocationBottom;
			END_IF
		(*Limit Y Location Top*)
			IF GV_Tool_Magazine.lrYLocationTop<GV_Tool_Magazine.lrMinYLocationTop THEN
				GV_Tool_Magazine.lrYLocationTop:=GV_Tool_Magazine.lrMinYLocationTop;
			END_IF
			IF GV_Tool_Magazine.lrYLocationTop>GV_Tool_Magazine.lrMaxYLocationTop THEN
				GV_Tool_Magazine.lrYLocationTop:=GV_Tool_Magazine.lrMaxYLocationTop;
			END_IF
		(*Limit Y Location Bottom*)
			IF GV_Tool_Magazine.lrYLocationBottom<GV_Tool_Magazine.lrMinYLocationBottom THEN
				GV_Tool_Magazine.lrYLocationBottom:=GV_Tool_Magazine.lrMinYLocationBottom;
			END_IF
			IF GV_Tool_Magazine.lrYLocationBottom>GV_Tool_Magazine.lrMaxYLocationBottom THEN
				GV_Tool_Magazine.lrYLocationBottom:=GV_Tool_Magazine.lrMaxYLocationBottom;
			END_IF
			
(** DATAS IN FUNCTION OF THE SETUP **)
	
	(* Infos Locations *) // aLocation
		FOR iLocationLoop:=1 TO GV_Tool_Magazine.iMaxAbsLocation BY 1 DO
			
			(*Number of the location in absolute*) // iAbsLocationNumber
				IF iLocationLoop<=GV_Tool_Magazine.iMaxRelLocation THEN
					GV_Tool_Magazine.aLocation[iLocationLoop].iAbsLocationNumber:=iLocationLoop;
				ELSE
					GV_Tool_Magazine.aLocation[iLocationLoop].iAbsLocationNumber:=0;
				END_IF
			
			(*Number of the location in relative*) // iRelLocationNumber
				IF iLocationLoop>2 AND iLocationLoop<=GV_Tool_Magazine.iMaxRelLocation THEN
					IF iLocationLoop<=GV_Tool_Magazine.iMaxRelLocationTop THEN
						GV_Tool_Magazine.aLocation[iLocationLoop].iRelLocationNumber:=iLocationLoop-2;
					ELSE
						IF iLocationLoop-GV_Tool_Magazine.iMaxRelLocationTop>1 THEN
						GV_Tool_Magazine.aLocation[iLocationLoop].iRelLocationNumber:=iLocationLoop-3;					
						ELSE
							GV_Tool_Magazine.aLocation[iLocationLoop].iRelLocationNumber:=0;
						END_IF
					END_IF
				ELSE
					GV_Tool_Magazine.aLocation[iLocationLoop].iRelLocationNumber:=0;
				END_IF	

			(*Number of the rack*) // iRackNumber
				IF iLocationLoop<=GV_Tool_Magazine.iMaxRelLocation THEN // same as : GV_Tool_Magazine.aLocation[iLocationLoop].iAbsLocationNumber=0
					FOR iRackLoop:=1 TO GV_Tool_Magazine.iMaxRelRack BY 1 DO			
						(*Top*)
							IF GV_Tool_Magazine.aLocation[iLocationLoop].iAbsLocationNumber>GV_Tool_Magazine.iMaxRelRackLocationTop*(iRackLoop-1) AND GV_Tool_Magazine.aLocation[iLocationLoop].iAbsLocationNumber<=GV_Tool_Magazine.iMaxRelRackLocationTop*(iRackLoop) AND GV_Tool_Magazine.aLocation[iLocationLoop].iAbsLocationNumber<=GV_Tool_Magazine.iMaxRelLocationTop THEN
								GV_Tool_Magazine.aLocation[iLocationLoop].iRackNumber:=iRackLoop;
							END_IF
						(*Bottom*)
							IF GV_Tool_Magazine.aLocation[iLocationLoop].iAbsLocationNumber>GV_Tool_Magazine.iMaxRelLocationTop AND GV_Tool_Magazine.aLocation[iLocationLoop].iAbsLocationNumber<=GV_Tool_Magazine.iMaxRelLocation THEN
								IF GV_Tool_Magazine.aLocation[iLocationLoop].iAbsLocationNumber-GV_Tool_Magazine.iMaxRelLocationTop>GV_Tool_Magazine.iMaxRelRackLocationBottom*(iRackLoop-1) AND GV_Tool_Magazine.aLocation[iLocationLoop].iAbsLocationNumber-GV_Tool_Magazine.iMaxRelLocationTop<=GV_Tool_Magazine.iMaxRelRackLocationBottom*(iRackLoop) THEN
									GV_Tool_Magazine.aLocation[iLocationLoop].iRackNumber:=iRackLoop+GV_Tool_Magazine.iMaxRelRackTop;
								END_IF
							END_IF
					END_FOR	
				ELSE
					GV_Tool_Magazine.aLocation[iLocationLoop].iRackNumber:=0;
				END_IF		
			
			(*Number of the location in the rack*) // iLocationRackNumber
				(*Top*)
					IF GV_Tool_Magazine.aLocation[iLocationLoop].iAbsLocationNumber=0 OR GV_Tool_Magazine.aLocation[iLocationLoop].iRackNumber=0 THEN
						GV_Tool_Magazine.aLocation[iLocationLoop].iLocationRackNumber:=0;
					END_IF
					IF GV_Tool_Magazine.aLocation[iLocationLoop].iRackNumber=1 THEN
						GV_Tool_Magazine.aLocation[iLocationLoop].iLocationRackNumber:=GV_Tool_Magazine.aLocation[iLocationLoop].iAbsLocationNumber;
					END_IF
					IF GV_Tool_Magazine.aLocation[iLocationLoop].iRackNumber>1 AND GV_Tool_Magazine.aLocation[iLocationLoop].iRackNumber<=GV_Tool_Magazine.iMaxRelRackTop THEN
						GV_Tool_Magazine.aLocation[iLocationLoop].iLocationRackNumber:=GV_Tool_Magazine.aLocation[iLocationLoop].iAbsLocationNumber-((GV_Tool_Magazine.aLocation[iLocationLoop].iRackNumber-1)*GV_Tool_Magazine.iMaxRelRackLocationTop);
					END_IF
				(*Bottom*)
					IF GV_Tool_Magazine.aLocation[iLocationLoop].iRackNumber>GV_Tool_Magazine.iMaxRelRackTop AND GV_Tool_Magazine.aLocation[iLocationLoop].iRackNumber<=GV_Tool_Magazine.iMaxRelRack THEN
						GV_Tool_Magazine.aLocation[iLocationLoop].iLocationRackNumber:=(GV_Tool_Magazine.aLocation[iLocationLoop].iAbsLocationNumber-GV_Tool_Magazine.iMaxRelLocationTop)-((GV_Tool_Magazine.aLocation[iLocationLoop].iRackNumber-GV_Tool_Magazine.iMaxRelRackTop-1)*GV_Tool_Magazine.iMaxRelRackLocationBottom);
					END_IF		
			
			(*Position of the location*) // ePositionMag
				IF GV_Tool_Magazine.aLocation[iLocationLoop].iRackNumber=0 THEN
					GV_Tool_Magazine.aLocation[iLocationLoop].ePositionMag:=ENUM_Position_Magazine.Unknow;			
				END_IF
				IF GV_Tool_Magazine.aLocation[iLocationLoop].iRackNumber>0 AND GV_Tool_Magazine.aLocation[iLocationLoop].iRackNumber<=GV_Tool_Magazine.iMaxRelRackTop THEN
					GV_Tool_Magazine.aLocation[iLocationLoop].ePositionMag:=ENUM_Position_Magazine.Top;
				END_IF
				IF GV_Tool_Magazine.aLocation[iLocationLoop].iRackNumber>GV_Tool_Magazine.iMaxRelRackTop AND GV_Tool_Magazine.aLocation[iLocationLoop].iRackNumber<=GV_Tool_Magazine.iMaxRelRack THEN
					GV_Tool_Magazine.aLocation[iLocationLoop].ePositionMag:=ENUM_Position_Magazine.Bottom;		
				END_IF
			
			(*Location enable*) // bEnable
				IF GV_Tool_Magazine.aLocation[iLocationLoop].iAbsLocationNumber>0 AND GV_Tool_Magazine.aLocation[iLocationLoop].iAbsLocationNumber<=GV_Tool_Magazine.iMaxRelLocation THEN
					GV_Tool_Magazine.aLocation[iLocationLoop].bEnable:=TRUE;
				ELSE
					GV_Tool_Magazine.aLocation[iLocationLoop].bEnable:=FALSE;
				END_IF
	
			(*Location used*) // bUsed
				IF GV_Tool_Magazine.aLocation[iLocationLoop].iAbsLocationNumber>0 AND GV_Tool_Magazine.aLocation[iLocationLoop].iAbsLocationNumber<=GV_Tool_Magazine.iMaxRelLocation THEN
					GV_Tool_Magazine.aLocation[iLocationLoop].bUsed:=TRUE;
				ELSE
					GV_Tool_Magazine.aLocation[iLocationLoop].bUsed:=FALSE;
				END_IF
			
			(*Location forbiden in absolute*) // bForbiden
				(*Top*)
					IF GV_Tool_Magazine.aLocation[iLocationLoop].iAbsLocationNumber=1 OR GV_Tool_Magazine.aLocation[iLocationLoop].iAbsLocationNumber=2 THEN
						GV_Tool_Magazine.aLocation[iLocationLoop].bForbiden:=TRUE;
					ELSE
						GV_Tool_Magazine.aLocation[iLocationLoop].bForbiden:=FALSE;		
					END_IF
				(*Bottom*)
					IF GV_Tool_Magazine.aLocation[iLocationLoop].iAbsLocationNumber>GV_Tool_Magazine.iMaxRelLocationTop THEN
						IF GV_Tool_Magazine.aLocation[iLocationLoop].iAbsLocationNumber-GV_Tool_Magazine.iMaxRelLocationTop=1 THEN
							GV_Tool_Magazine.aLocation[iLocationLoop].bForbiden:=TRUE;
						ELSE
							GV_Tool_Magazine.aLocation[iLocationLoop].bForbiden:=FALSE;			
						END_IF
					END_IF
			
			(*Location Tool*)
				(*Presence*) // bToolPresence (*Breakage ctrl*) // bBreakageOk
					IF GV_Tool_Magazine.aLocation[iLocationLoop].iRelLocationNumber<>0 THEN
						GV_Tool_Magazine.aLocation[iLocationLoop].bToolPresence:=TRUE;
						GV_Tool_Magazine.aLocation[iLocationLoop].bBreakageOk:=TRUE;
					ELSE
						GV_Tool_Magazine.aLocation[iLocationLoop].bToolPresence:=FALSE;
						GV_Tool_Magazine.aLocation[iLocationLoop].bBreakageOk:=FALSE;
					END_IF
	
					IF GV_Tool_Magazine.aLocation[iLocationLoop].iAbsLocationNumber=0 THEN
						GV_Tool_Magazine.aLocation[iLocationLoop].eToolType:=ENUM_Tool_Type.Unknow;
						GV_Tool_Magazine.aLocation[iLocationLoop].bToolPresence:=FALSE;
						
						GV_Tool_Magazine.aLocation[iLocationLoop].stToolParam:=GV_Tool_Magazine.stEmptyToolParam;
						GV_Tool_Magazine.aLocation[iLocationLoop].stToolName:=GV_Tool_Magazine.stEmptyToolName;
					END_IF
			
			(*X,Y coordinate*) // lrXcoord and lrYcoord
				//IF GV_Tool_Magazine.aLocation[iLocationLoop].iAbsLocationNumber=0 THEN
				//	GV_Tool_Magazine.aLocation[iLocationLoop].lrXcoord:=0;
				//	GV_Tool_Magazine.aLocation[iLocationLoop].lrYcoord:=0;
				//END_IF
				(*Top*)
					//IF GV_Tool_Magazine.aLocation[iLocationLoop].iAbsLocationNumber>0 AND GV_Tool_Magazine.aLocation[iLocationLoop].iAbsLocationNumber<=GV_Tool_Magazine.iMaxRelLocationTop THEN
					//	GV_Tool_Magazine.aLocation[iLocationLoop].lrXcoord:=GV_Tool_Magazine.lrXFirstLocationTop+(GV_Tool_Magazine.lrXLocationOffsetTop*(GV_Tool_Magazine.iMaxRelRackLocationTop-GV_Tool_Magazine.aLocation[iLocationLoop].iLocationRackNumber));
					//	GV_Tool_Magazine.aLocation[iLocationLoop].lrYcoord:=GV_Tool_Magazine.lrYLocationOffsetTop;
					//END_IF
				(*Bottom*)
					//IF GV_Tool_Magazine.aLocation[iLocationLoop].iAbsLocationNumber>GV_Tool_Magazine.iMaxRelLocationTop AND GV_Tool_Magazine.aLocation[iLocationLoop].iAbsLocationNumber<=GV_Tool_Magazine.iMaxRelLocation THEN
					//	GV_Tool_Magazine.aLocation[iLocationLoop].lrXcoord:=GV_Tool_Magazine.lrXFirstLocationBottom+(GV_Tool_Magazine.lrXLocationOffsetBottom*(GV_Tool_Magazine.iMaxRelRackLocationBottom-GV_Tool_Magazine.aLocation[iLocationLoop].iLocationRackNumber));			
					//	GV_Tool_Magazine.aLocation[iLocationLoop].lrYcoord:=GV_Tool_Magazine.lrYLocationOffsetBottom;
					//END_IF 		
			(*Z coordinate*) // lrZcoord
				//IF GV_Tool_Magazine.aLocation[iLocationLoop].iAbsLocationNumber=0 THEN
				//	GV_Tool_Magazine.aLocation[iLocationLoop].lrZcoord:=0;
				//END_IF
				(*Top*)
					//IF GV_Tool_Magazine.aLocation[iLocationLoop].iRackNumber>0 AND GV_Tool_Magazine.aLocation[iLocationLoop].iRackNumber<=GV_Tool_Magazine.iMaxRelRackTop THEN
					//	GV_Tool_Magazine.aLocation[iLocationLoop].lrZcoord:=GV_Tool_Magazine.lrZLowestRackTop+(GV_Tool_Magazine.lrZLocationOffsetTop*(GV_Tool_Magazine.aLocation[iLocationLoop].iRackNumber-1));
					//	GV_Tool_Magazine.aLocation[iLocationLoop].lrZcoord:=GV_Tool_Magazine.aLocation[iLocationLoop].lrZcoord-(GV_Tool_Magazine.lrZRelCompensationLocationTop*(GV_Tool_Magazine.iMaxRelRackLocationTop-GV_Tool_Magazine.aLocation[iLocationLoop].iLocationRackNumber));// Compensation
					//END_IF			
				(*Bottom*)
					//IF GV_Tool_Magazine.aLocation[iLocationLoop].iRackNumber>GV_Tool_Magazine.iMaxRelRackTop AND GV_Tool_Magazine.aLocation[iLocationLoop].iRackNumber<=GV_Tool_Magazine.iMaxRelRack THEN
					//	GV_Tool_Magazine.aLocation[iLocationLoop].lrZcoord:=GV_Tool_Magazine.lrZLowestRackBottom+(GV_Tool_Magazine.lrZLocationOffsetBottom*(GV_Tool_Magazine.iMaxRelRack-GV_Tool_Magazine.aLocation[iLocationLoop].iRackNumber));
					//	GV_Tool_Magazine.aLocation[iLocationLoop].lrZcoord:=GV_Tool_Magazine.aLocation[iLocationLoop].lrZcoord-(GV_Tool_Magazine.lrZRelCompensationLocationBottom*(GV_Tool_Magazine.iMaxRelRackLocationBottom-GV_Tool_Magazine.aLocation[iLocationLoop].iLocationRackNumber));// Compensation
					//END_IF
			
			(*X,Y,Z coordinate*) // lrXcoord lrYcoord lrZcoord
				IF GV_Tool_Magazine.aLocation[iLocationLoop].ePositionMag=ENUM_Position_Magazine.Top THEN
					GV_Tool_Magazine.aLocation[iLocationLoop].lrXcoord:=GV_Tool_Magazine.lrXFirstLocationTop+(GV_Tool_Magazine.lrXLocationOffsetTop*(GV_Tool_Magazine.aLocation[iLocationLoop].iLocationRackNumber-1));
						GV_Tool_Magazine.aLocation[iLocationLoop].lrXcoord:=LINT_TO_LREAL(LREAL_TO_LINT(GV_Tool_Magazine.aLocation[iLocationLoop].lrXcoord*1000.0))/1000.0; // Round 10e-3 (normally not usefull)
					GV_Tool_Magazine.aLocation[iLocationLoop].lrYcoord:=GV_Tool_Magazine.lrYLocationTop+(GV_Tool_Magazine.lrYLocationOffsetTop*(GV_Tool_Magazine.aLocation[iLocationLoop].iLocationRackNumber-1));
						GV_Tool_Magazine.aLocation[iLocationLoop].lrYcoord:=LINT_TO_LREAL(LREAL_TO_LINT(GV_Tool_Magazine.aLocation[iLocationLoop].lrYcoord*1000.0))/1000.0; // Round 10e-3 (normally not usefull)					
					GV_Tool_Magazine.aLocation[iLocationLoop].lrZcoord:=GV_Tool_Magazine.lrZLowestRackTop+(GV_Tool_Magazine.lrZLocationOffsetTop*(GV_Tool_Magazine.aLocation[iLocationLoop].iRackNumber-1));
					GV_Tool_Magazine.aLocation[iLocationLoop].lrZcoord:=GV_Tool_Magazine.aLocation[iLocationLoop].lrZcoord-(GV_Tool_Magazine.lrZRelCompensationLocationTop*(GV_Tool_Magazine.aLocation[iLocationLoop].iLocationRackNumber));// Compensation
						GV_Tool_Magazine.aLocation[iLocationLoop].lrZcoord:=LINT_TO_LREAL(LREAL_TO_LINT(GV_Tool_Magazine.aLocation[iLocationLoop].lrZcoord*1000.0))/1000.0; // Round 10e-3
				ELSIF GV_Tool_Magazine.aLocation[iLocationLoop].ePositionMag=ENUM_Position_Magazine.Bottom THEN
					GV_Tool_Magazine.aLocation[iLocationLoop].lrXcoord:=GV_Tool_Magazine.lrXFirstLocationBottom+(GV_Tool_Magazine.lrXLocationOffsetBottom*(GV_Tool_Magazine.aLocation[iLocationLoop].iLocationRackNumber-1));
						GV_Tool_Magazine.aLocation[iLocationLoop].lrXcoord:=LINT_TO_LREAL(LREAL_TO_LINT(GV_Tool_Magazine.aLocation[iLocationLoop].lrXcoord*1000.0))/1000.0; // Round 10e-3 (normally not usefull)
					GV_Tool_Magazine.aLocation[iLocationLoop].lrYcoord:=GV_Tool_Magazine.lrYLocationBottom+(GV_Tool_Magazine.lrYLocationOffsetBottom*(GV_Tool_Magazine.aLocation[iLocationLoop].iLocationRackNumber-1));
						GV_Tool_Magazine.aLocation[iLocationLoop].lrYcoord:=LINT_TO_LREAL(LREAL_TO_LINT(GV_Tool_Magazine.aLocation[iLocationLoop].lrYcoord*1000.0))/1000.0; // Round 10e-3 (normally not usefull)					
					GV_Tool_Magazine.aLocation[iLocationLoop].lrZcoord:=GV_Tool_Magazine.lrZLowestRackBottom+(GV_Tool_Magazine.lrZLocationOffsetBottom*(GV_Tool_Magazine.iMaxRelRack-GV_Tool_Magazine.aLocation[iLocationLoop].iRackNumber));//(GV_Tool_Magazine.aLocation[iLocationLoop].iRackNumber-1));
					GV_Tool_Magazine.aLocation[iLocationLoop].lrZcoord:=GV_Tool_Magazine.aLocation[iLocationLoop].lrZcoord-(GV_Tool_Magazine.lrZRelCompensationLocationBottom*(GV_Tool_Magazine.aLocation[iLocationLoop].iLocationRackNumber));// Compensation
						GV_Tool_Magazine.aLocation[iLocationLoop].lrZcoord:=LINT_TO_LREAL(LREAL_TO_LINT(GV_Tool_Magazine.aLocation[iLocationLoop].lrZcoord*1000.0))/1000.0; // Round 10e-3
				ELSE
					GV_Tool_Magazine.aLocation[iLocationLoop].lrXcoord:=0;
					GV_Tool_Magazine.aLocation[iLocationLoop].lrYcoord:=0;
					GV_Tool_Magazine.aLocation[iLocationLoop].lrZcoord:=0;
				END_IF
			
		END_FOR

END_PROGRAM

// ---- 09_Tool_Magazine/03_POUs/01_PRGs/PRG_Tool_Magazine_Type1.TcPOU
PROGRAM PRG_Tool_Magazine_Type1
VAR
	(** ENUM **)
		(*Manipulator Gripper mvmnt*)
			eGripperMode : ENUM_Gripper_Mode; // Gripper mode for gripper mouvement (fbGripper)

	(** TIME **)
		(*Manipulator Gripper mvmnt*)
			tGripperTime : TIME ; // Mouvement duration for gripper mouvement (fbGripper)

	(** LREAL **)
		lrTeachRackZ : LREAL := 0.0 ; // Z for Teach Rack
		lrTeachAllX : LREAL := 0.0 ; // X for Teach All
		lrTeachAllY : LREAL := 0.0 ; // Y for Teach All
		lrTeachAllZ : LREAL := 0.0 ; // Z for Teach All
		
	(** INT **)
		iRackLoop : INT := 0 ; // Use in a FOR Loop
		iLocationLoop : INT := 0 ; // Use in a FOR Loop
		iCheckLocationLoop : INT := 0 ; // Use in a FOR Loop
		iTeachLoop : INT := 0 ; // Use in a FOR Loop
		iCount : INT := 0 ; // Use for count in a FOR Loop
		
	(** FLAG **)
		(*Manipulator Gripper mvmnt*)
			bGripperSensor : BOOL ; // Sensor check for gripper mouvement (fbGripper)
	
	(** FB **)
		fbReverseToolLocation : FB_ArrayToolLocation_Reverse ;
		fbGripperManu : FB_Manipulator_Gripper ;
END_VAR

//-----------------------------------------------------------------------------------------
//
//                  		PRG_Tool_Magazine_Type1
//
//					Gestion magasin outils durant le cycle		
//-----------------------------------------------------------------------------------------
//
//Auteur: G.GOETZ
//Création: 14.01.2026
//Dernière modification : 14.01.2026 (G.GOETZ)
//       			
//-----------------------------------------------------------------------------------------
//
//     							Liste des modifications  	
//
// 14.01.2026 (G.GOETZ) -> Création		
//-----------------------------------------------------------------------------------------

(** DATAS **)

	(** Check Location ordering**)
		IF GV_Tool_Magazine.bFullCheckMagazineInitLocation THEN
			GV_Tool_Magazine.iCheckLocationTopSize:=0;
			GV_Tool_Magazine.iCheckLocationBottomSize:=0;
			FOR iCheckLocationLoop:=1 TO GV_Tool_Magazine.iMaxAbsLocation BY 1 DO
				GV_Tool_Magazine.aCheckLocation[iCheckLocationLoop]:=GV_Tool_Magazine.stEmptyToolLocation;
			END_FOR
		END_IF

	(* Infos Locations *) // aLocation
		FOR iLocationLoop:=1 TO GV_Tool_Magazine.iMaxAbsLocation BY 1 DO

			(*Tool presence*) // bToolPresence
				//IF GV_Tool_Magazine.aLocation[iLocationLoop].stToolParam.Number<>0 THEN
				//	GV_Tool_Magazine.aLocation[iLocationLoop].bToolPresence:=TRUE;
				//ELSE
				//	GV_Tool_Magazine.aLocation[iLocationLoop].bToolPresence:=FALSE;		
				//END_IF
			
			(*Tool type*)// eToolType
				//IF GV_Tool_Magazine.aLocation[iLocationLoop].bToolPresence THEN //  -> Revoir la philosophie
					IF GV_Tool_Magazine.aLocation[iLocationLoop].stToolParam.Size=1 OR TRUE THEN
						GV_Tool_Magazine.aLocation[iLocationLoop].eToolType:=ENUM_Tool_Type.Small;
					ELSIF GV_Tool_Magazine.aLocation[iLocationLoop].stToolParam.Size=2 THEN
						GV_Tool_Magazine.aLocation[iLocationLoop].eToolType:=ENUM_Tool_Type.Big;
					ELSIF GV_Tool_Magazine.aLocation[iLocationLoop].stToolParam.Size=3 THEN
						GV_Tool_Magazine.aLocation[iLocationLoop].eToolType:=ENUM_Tool_Type.Big;
					ELSE
						GV_Tool_Magazine.aLocation[iLocationLoop].eToolType:=ENUM_Tool_Type.Unknow;
					END_IF
				//ELSE
				//	GV_Tool_Magazine.aLocation[iLocationLoop].eToolType:=ENUM_Tool_Type.Unknow;
				//END_IF
			
			(*Location blocked*) // bBlocked
				IF GV_Tool_Magazine.aLocation[iLocationLoop].iAbsLocationNumber>1 THEN
					IF GV_Tool_Magazine.aLocation[iLocationLoop-1].bBlocked=FALSE AND GV_Tool_Magazine.aLocation[iLocationLoop-1].iRackNumber=GV_Tool_Magazine.aLocation[iLocationLoop].iRackNumber AND (GV_Tool_Magazine.aLocation[iLocationLoop-1].eToolType=ENUM_Tool_Type.Big OR GV_Tool_Magazine.aLocation[iLocationLoop-1].eToolType=ENUM_Tool_Type.GPS70) THEN
						GV_Tool_Magazine.aLocation[iLocationLoop].bBlocked:=TRUE;
					ELSE
						GV_Tool_Magazine.aLocation[iLocationLoop].bBlocked:=FALSE;
					END_IF
				ELSE
					GV_Tool_Magazine.aLocation[iLocationLoop].bBlocked:=FALSE;
				END_IF
				
			(** Check Location ordering**)
				IF GV_Tool_Magazine.bFullCheckMagazineInitLocation THEN
					FOR iCheckLocationLoop:=1 TO GV_Tool_Magazine.iMaxAbsLocation BY 1 DO
						IF GV_Tool_Magazine.aCheckLocation[iCheckLocationLoop].iRelLocationNumber=0 AND GV_Tool_Magazine.aLocation[iLocationLoop].iRelLocationNumber<>0 THEN
							IF GV_Tool_Magazine.aLocation[iLocationLoop].ePositionMag=ENUM_Position_Magazine.Top THEN
								GV_Tool_Magazine.aCheckLocation[iCheckLocationLoop]:=GV_Tool_Magazine.aLocation[iLocationLoop];
								GV_Tool_Magazine.iCheckLocationTopSize:=GV_Tool_Magazine.iCheckLocationTopSize+1;
							ELSIF GV_Tool_Magazine.aLocation[iLocationLoop].ePositionMag=ENUM_Position_Magazine.Bottom THEN
								GV_Tool_Magazine.aCheckLocation[iCheckLocationLoop]:=GV_Tool_Magazine.aLocation[iLocationLoop];
								GV_Tool_Magazine.iCheckLocationBottomSize:=GV_Tool_Magazine.iCheckLocationBottomSize+1;
							END_IF
							EXIT; // Stop For Loop
						//ELSE
						//	GV_Tool_Magazine.aCheckLocation[iCheckLocationLoop]:=GV_Tool_Magazine.stEmptyToolLocation;
						END_IF
					END_FOR
				END_IF
				
		END_FOR
		(* Reverse Location*)
		IF GV_Tool_Magazine.bFullCheckMagazineInitLocation THEN
			fbReverseToolLocation(
									aArray:=GV_Tool_Magazine.aCheckLocation,
									iHighSize:=GV_Tool_Magazine.iCheckLocationTopSize,
									iLowSize:=GV_Tool_Magazine.iCheckLocationBottomSize,
									bReverseHigh:=TRUE,
									bReverseLow:=TRUE,
									bReverseRowHigh:=TRUE,
									bReverseRowLow:=TRUE
									);
		END_IF
		GV_Tool_Magazine.bFullCheckMagazineInitLocation:=FALSE;
		
(** MANIPULATOR HEAD **)
	(*Axis Position*)
		GV_Tool_Magazine.stManipulator.lrXPosition:=LINT_TO_LREAL(LREAL_TO_LINT(GV_Axes.stAxisX.stDriveAx8206.AxisRef.NcToPlc.ActPos*1000.0))/1000.0;
		GV_Tool_Magazine.stManipulator.lrYPosition:=LINT_TO_LREAL(LREAL_TO_LINT(GV_Axes.stAxisY.stDriveAx8206.AxisRef.NcToPlc.ActPos*1000.0))/1000.0;
		GV_Tool_Magazine.stManipulator.lrZPosition:=LINT_TO_LREAL(LREAL_TO_LINT(GV_Axes.stAxisZ.stDriveAx8206.AxisRef.NcToPlc.ActPos*1000.0))/1000.0;
	(*Memory*)
		IF (GV_Tool_Magazine.stManipulator.iAbsLocationNumberMemory<>0 AND GV_Tool_Magazine.stManipulator.iRelLocationNumberMemory<>0) THEN
			GV_Tool_Magazine.stManipulator.bToolPresenceMemory:=TRUE;
		ELSE
			GV_Tool_Magazine.stManipulator.bToolPresenceMemory:=FALSE;
		END_IF
	(*PositionMag*)
		IF GV_Tool_Magazine.stManipulator.lrZPosition>=500 THEN //GV_Tool_Magazine.lrZLowestRackTop-1(*GV_Tool_Magazine.stManipulator.lrZTunnelTop*) THEN
			GV_Tool_Magazine.stManipulator.ePositionMag:=ENUM_Position_Magazine.Top;
		ELSIF GV_Tool_Magazine.stManipulator.lrZPosition<=GV_Tool_Magazine.stManipulator.lrZTunnelBottom THEN
			GV_Tool_Magazine.stManipulator.ePositionMag:=ENUM_Position_Magazine.Bottom;
		ELSE
			GV_Tool_Magazine.stManipulator.ePositionMag:=ENUM_Position_Magazine.Unknow;
		END_IF
	(*Positions*)	
		IF GV_Tool_Magazine.stManipulator.lrXPosition<=(GV_Tool_Magazine.stManipulator.lrXHome+GV_Tool_Magazine.stManipulator.lrXPositionTol) AND GV_Tool_Magazine.stManipulator.lrXPosition>=(GV_Tool_Magazine.stManipulator.lrXHome-GV_Tool_Magazine.stManipulator.lrXPositionTol) AND // X
		   GV_Tool_Magazine.stManipulator.lrYPosition<=(GV_Tool_Magazine.stManipulator.lrYHome+GV_Tool_Magazine.stManipulator.lrYPositionTol) AND GV_Tool_Magazine.stManipulator.lrYPosition>=(GV_Tool_Magazine.stManipulator.lrYHome-GV_Tool_Magazine.stManipulator.lrYPositionTol) AND // Y
		   GV_Tool_Magazine.stManipulator.lrZPosition<=(GV_Tool_Magazine.stManipulator.lrZHome+GV_Tool_Magazine.stManipulator.lrZPositionTol) AND GV_Tool_Magazine.stManipulator.lrZPosition>=(GV_Tool_Magazine.stManipulator.lrZHome-GV_Tool_Magazine.stManipulator.lrZPositionTol) THEN // Z
			GV_Tool_Magazine.stManipulator.ePositionAxis:=ENUM_Position_Axis.Home;
		//ELSIF
		ELSE
			GV_Tool_Magazine.stManipulator.ePositionAxis:=ENUM_Position_Axis.Unknow;
		END_IF
		(*YTunnel=YHome*)
			GV_Tool_Magazine.stManipulator.lrYTunnel:=GV_Tool_Magazine.stManipulator.lrYHome;
	(*Exclusion Zones*)
		
	
	(*Close/Clamp Gripper Manual Authorization*)
		IF GV_OpMode.eOpMode=ENUM_OpMode.MANU AND GV_General.bSafety AND GV_General.bPower AND GV_General.bAir AND (*xxx AND *) (NOT fbGripperManu.bStart) AND (NOT fbGripperManu.bBusy) THEN
			GV_Tool_Magazine.stManipulator.bAuthorizationManuGripperClose:=TRUE; ;
		ELSE
			GV_Tool_Magazine.stManipulator.bAuthorizationManuGripperClose:=FALSE;
		END_IF
	(*Close/Clamp Gripper Manual Command*)
		IF GV_Tool_Magazine.stManipulator.bAuthorizationManuGripperClose AND GV_HMI.stManipulatorGripper.rtCloseManupulatorGripper.Q THEN
			eGripperMode:=ENUM_Gripper_Mode.Close; // Gripper mode
			tGripperTime:=GV_HMI.stManipulatorGripper.tMouvementClose; // Gripper mouvement time
			bGripperSensor:=FALSE; //GV_HMI.stManipulatorGripper.bCheckSensorOpen; // Gripper check sensor
			fbGripperManu.bStart:=TRUE; // Gripper Start
			(*Log*)
				PRG_Log_WM.fbLogWM.M_Write_Log('MANUAL : GripperClamp -> SATRT');
		END_IF
	(*Open/Unclamp Gripper Manual Authorization*)
		IF GV_OpMode.eOpMode=ENUM_OpMode.MANU AND GV_General.bSafety AND GV_General.bPower AND GV_General.bAir AND (*xxx AND *) (NOT fbGripperManu.bStart) AND (NOT fbGripperManu.bBusy) THEN
			GV_Tool_Magazine.stManipulator.bAuthorizationManuGripperOpen:=TRUE;
		ELSE
			GV_Tool_Magazine.stManipulator.bAuthorizationManuGripperOpen:=FALSE;
		END_IF
	(*Open/Unclamp Gripper Manual Command*)
		IF GV_Tool_Magazine.stManipulator.bAuthorizationManuGripperOpen AND GV_HMI.stManipulatorGripper.rtOpenManupulatorGripper.Q THEN
			eGripperMode:=ENUM_Gripper_Mode.Open; // Gripper mode
			tGripperTime:=GV_HMI.stManipulatorGripper.tMouvementOpen; // Gripper mouvement time
			bGripperSensor:=FALSE; //GV_HMI.stManipulatorGripper.bCheckSensorClose; // Gripper check sensor
			fbGripperManu.bStart:=TRUE; // Gripper Start
			(*Log*)
				PRG_Log_WM.fbLogWM.M_Write_Log('MANUAL : GripperUnclamp -> SATRT');
		END_IF
		
